	FB_SelectArray(sNetID:= , hDBID:= 1, cbCmdSize:= SIZEOF(GVL_DB.slctAllMethods), pCmdAddr:= ADR(GVL_DB.slctAllMethods), nStartIndex:= 0, nRecordCount:= 500, cbRecordArraySize:= SIZEOF(GVL_DB.listOfMethod), pDestAddr:= ADR(GVL_DB.listOfMethod), bExecute:= TRUE, tTimeout:= T#15S, bBusy=> busy, bError=> err, nErrID=> errid, sSQLState=> sqlstate, nRecords=> recAnz);
	
	IF NOT FB_SelectArray.bBusy THEN
		state:= E_DB_QUERY_STATE.IDLE_STATE;
		bExecute:= FALSE;
	ELSIF FB_SelectArray.bError THEN	
		state:= E_DB_QUERY_STATE.ERROR_STATE;
	ELSE
		state:= E_DB_QUERY_STATE.SELECT_ALL_METHODS;
		bExecute:= FALSE;
	END_IF
	
E_DB_QUERY_STATE.SELECT_ALL_ACTV_METHODS:
	
	FB_SelectArray(sNetID:= , hDBID:= 1, cbCmdSize:= SIZEOF(GVL_DB.slctAllActvMethod), pCmdAddr:= ADR(GVL_DB.slctAllActvMethod), nStartIndex:= 0, nRecordCount:= 500, cbRecordArraySize:= SIZEOF(GVL_DB.listOfMethod), pDestAddr:= ADR(GVL_DB.listOfMethod), bExecute:= TRUE, tTimeout:= T#15S, bBusy=> busy, bError=> err, nErrID=> errid, sSQLState=> sqlstate, nRecords=> recAnz);
	
	IF NOT FB_SelectArray.bBusy THEN
		state:= E_DB_QUERY_STATE.IDLE_STATE;
		bExecute:= FALSE;
	ELSIF FB_SelectArray.bError THEN	
		state:= E_DB_QUERY_STATE.ERROR_STATE;
	ELSE
		state:= E_DB_QUERY_STATE.SELECT_ALL_ACTV_METHODS;
		bExecute:= FALSE;
	END_IF
	
E_DB_QUERY_STATE.SELECT_WHOLE_METHODS:
	
	cmdSlc:= GVL_DB.slctMethod;
	selectMethod(start:=TRUE, methodName:= GVL_DB.methodName, methodRevision:= GVL_DB.methodRevision);
	FB_SelectArray(sNetID:= , hDBID:= 1, cbCmdSize:= SIZEOF(cmdSlc), pCmdAddr:= ADR(cmdSlc), nStartIndex:= 0, nRecordCount:= 26, cbRecordArraySize:= SIZEOF(GVL_DB.stParameter_MR), pDestAddr:= ADR(GVL_DB.stParameter_MR), bExecute:= TRUE, tTimeout:= T#15S, bBusy=> busy, bError=> err, nErrID=> errid, sSQLState=> sqlstate, nRecords=> recAnz);
	
	IF NOT FB_SelectArray.bBusy THEN
		timerVD(in:= TRUE, pt:= T#3S);
		bExecute:= FALSE;
		state:= E_DB_QUERY_STATE.IDLE_STATE;
	ELSIF FB_SelectArray.bError THEN	
		state:= E_DB_QUERY_STATE.ERROR_STATE;
	ELSE
		state:= E_DB_QUERY_STATE.SELECT_WHOLE_METHODS;
		bExecute:= FALSE;
	END_IF
	
E_DB_QUERY_STATE.INSERT_NEW_METHOD:

	cmdIn:= GVL_DB.isrtNewMethod;
	insertMethod(start:=TRUE);
	FB_Insert(sNetID:= , hDBID:= 1, cbCmdSize:= SIZEOF(cmdIn), pCmdAddr:= ADR(cmdIn), bExecute:= TRUE, tTimeout:= T#15S, bBusy=> busy, bError=> err, nErrID=> errid, sSQLState=> sqlstate);
	
	IF NOT FB_Insert.bBusy THEN
		state:= E_DB_QUERY_STATE.IDLE_STATE;
		bExecuteIn:= FALSE;
	ELSIF FB_Insert.bError THEN	
		state:= E_DB_QUERY_STATE.ERROR_STATE;
	ELSE
		state:= E_DB_QUERY_STATE.INSERT_NEW_METHOD;
		//bExecuteIn:= FALSE;
	END_IF	

E_DB_QUERY_STATE.UPDATE_DEACTV_METHOD:

	cmdIn:= GVL_DB.updtDactvMethod;
	updateMethod(start:=TRUE, methodName:= GVL_Recipe.stCurrentRecipe.stInfo.sMethodName, methodRevision:= INT_TO_STRING(GVL_Recipe.stCurrentRecipe.stInfo.iRevision));
	FB_Insert(sNetID:= , hDBID:= 1, cbCmdSize:= SIZEOF(cmdIn), pCmdAddr:= ADR(cmdIn), bExecute:= TRUE, tTimeout:= T#15S, bBusy=> busy, bError=> err, nErrID=> errid, sSQLState=> sqlstate);
	
	IF NOT FB_Insert.bBusy THEN
		state:= E_DB_QUERY_STATE.IDLE_STATE;
		bExecuteIn:= FALSE;
	ELSIF FB_Insert.bError THEN	
		state:= E_DB_QUERY_STATE.ERROR_STATE;
	ELSE
		state:= E_DB_QUERY_STATE.UPDATE_DEACTV_METHOD;
		//bExecuteIn:= FALSE;
	END_IF	

E_DB_QUERY_STATE.SELECT_LAST_METHOD_ID:
	
	cmdSlc:= GVL_DB.slctMethodID;
	selectMethodID(start:= TRUE, methodName:= GVL_HMI.stRecipeInfo.sMethodName);
	FB_SelectArray(sNetID:= , hDBID:= 1, cbCmdSize:= SIZEOF(cmdSlc), pCmdAddr:= ADR(cmdSlc), nStartIndex:= 0, nRecordCount:= 1, cbRecordArraySize:= SIZEOF(GVL_DB.lastMethodID), pDestAddr:= ADR(GVL_DB.lastMethodID), bExecute:= TRUE, tTimeout:= T#15S, bBusy=> busy, bError=> err, nErrID=> errid, sSQLState=> sqlstate, nRecords=> recAnz);
	
	IF NOT FB_SelectArray.bBusy THEN
		state:= E_DB_QUERY_STATE.IDLE_STATE;
		bExecute:= FALSE;
	ELSIF FB_SelectArray.bError THEN	
		state:= E_DB_QUERY_STATE.ERROR_STATE;
	ELSE
		state:= E_DB_QUERY_STATE.SELECT_LAST_METHOD_ID;
		bExecute:= FALSE;
	END_IF
	
E_DB_QUERY_STATE.SELECT_VOLUME_DATA:
	
	cmdSlc:= GVL_DB.slctVD;
	selectVD(start:=TRUE, methodID:= INT_TO_STRING(GVL_DB.stParameter_MR.methodID));
	FB_SelectArray(sNetID:= , hDBID:= 1, cbCmdSize:= SIZEOF(cmdSlc), pCmdAddr:= ADR(cmdSlc), nStartIndex:= 0, nRecordCount:= 10, cbRecordArraySize:= SIZEOF(GVL_DB.astVolData), pDestAddr:= ADR(GVL_DB.astVolData), bExecute:= TRUE, tTimeout:= T#15S, bBusy=> busy, bError=> err, nErrID=> errid, sSQLState=> sqlstate, nRecords=> recAnz);
	
	IF NOT FB_SelectArray.bBusy AND timerVD.Q THEN
		state:= E_DB_QUERY_STATE.IDLE_STATE;
		bExecute:= FALSE;
		//timerVD(in:= FALSE);
	ELSIF FB_SelectArray.bError THEN	
		state:= E_DB_QUERY_STATE.ERROR_STATE;
	ELSE
		state:= E_DB_QUERY_STATE.SELECT_VOLUME_DATA;
		bExecute:= FALSE;
	END_IF
	
E_DB_QUERY_STATE.INSERT_VOLUME_DATA:

	cmdIn:= GVL_DB.isrtVD;
	insertVD(start:=TRUE, methodID:= INT_TO_STRING(GVL_DB.lastMethodID), line:= j);
	FB_Insert(sNetID:= , hDBID:= 1, cbCmdSize:= SIZEOF(cmdIn), pCmdAddr:= ADR(cmdIn), bExecute:= TRUE, tTimeout:= T#15S, bBusy=> busy, bError=> err, nErrID=> errid, sSQLState=> sqlstate);
	
	IF NOT FB_Insert.bBusy THEN
		state:= E_DB_QUERY_STATE.IDLE_STATE;
		bExecuteIn:= FALSE;
	ELSIF FB_Insert.bError THEN	
		state:= E_DB_QUERY_STATE.ERROR_STATE;
	ELSE
		state:= E_DB_QUERY_STATE.INSERT_VOLUME_DATA;
		//bExecuteIn:= FALSE;
	END_IF	
	
E_DB_QUERY_STATE.INSERT_USER:

    cmdIn := GVL_DB.isrtUser;
    insertUser(start := TRUE, line := i);

    FB_Insert(
        sNetID := ,
        hDBID := 1,
        cbCmdSize := SIZEOF(cmdIn),
        pCmdAddr := ADR(cmdIn),
        bExecute := TRUE,
        tTimeout := T#15S,
        bBusy => busy,
        bError => err,
        nErrID => errid,
        sSQLState => sqlstate
    );

    IF NOT FB_Insert.bBusy THEN
        state := E_DB_QUERY_STATE.IDLE_STATE;
        bExecuteIn := FALSE;
    ELSIF FB_Insert.bError THEN
        state := E_DB_QUERY_STATE.ERROR_STATE;
    ELSE
        state := E_DB_QUERY_STATE.INSERT_USER;
    END_IF
(*	
E_DB_QUERY_STATE.INSERT_USER_MGMT_HISTORY:

    cmdIn := GVL_DB.isrtUserMgmtHistory;
    insertUserMgmtHistory(start := TRUE);

    GVL_HMI.stUserMgmtHistoryEvent.bBusy := TRUE;
    GVL_HMI.stUserMgmtHistoryEvent.bDone := FALSE;
    GVL_HMI.stUserMgmtHistoryEvent.bError := FALSE;
    GVL_HMI.stUserMgmtHistoryEvent.sErrorText := '';

    FB_Insert(
        sNetID := ,
        hDBID := 1,
        cbCmdSize := SIZEOF(cmdIn),
        pCmdAddr := ADR(cmdIn),
        bExecute := TRUE,
        tTimeout := T#15S,
        bBusy => busy,
        bError => err,
        nErrID => errid,
        sSQLState => sqlstate
    );

    IF NOT FB_Insert.bBusy THEN

        GVL_HMI.stUserMgmtHistoryEvent.bExecute := FALSE;
        GVL_HMI.stUserMgmtHistoryEvent.bBusy := FALSE;
        GVL_HMI.stUserMgmtHistoryEvent.bDone := TRUE;
        GVL_HMI.stUserMgmtHistoryEvent.bError := FALSE;

        state := E_DB_QUERY_STATE.IDLE_STATE;
        bExecuteIn := FALSE;

    ELSIF FB_Insert.bError THEN

        GVL_HMI.stUserMgmtHistoryEvent.bExecute := FALSE;
        GVL_HMI.stUserMgmtHistoryEvent.bBusy := FALSE;
        GVL_HMI.stUserMgmtHistoryEvent.bDone := FALSE;
        GVL_HMI.stUserMgmtHistoryEvent.bError := TRUE;
        GVL_HMI.stUserMgmtHistoryEvent.sErrorText := 'Error inserting user management history.';

        state := E_DB_QUERY_STATE.ERROR_STATE;

    ELSE

        state := E_DB_QUERY_STATE.INSERT_USER_MGMT_HISTORY;
        bExecuteIn := FALSE;

    END_IF
*)
E_DB_QUERY_STATE.SELECT_ALL_CURRENT_USERS:
	
	cmdSlc:= GVL_DB.slctCurrentUser;
	FB_SelectArray(sNetID:= , hDBID:= 1, cbCmdSize:= SIZEOF(cmdSlc), pCmdAddr:= ADR(cmdSlc), nStartIndex:= 0, nRecordCount:= 500, cbRecordArraySize:= SIZEOF(GVL_DB.astData_CUL), pDestAddr:= ADR(GVL_DB.astData_CUL), bExecute:= TRUE, tTimeout:= T#15S, bBusy=> busy, bError=> err, nErrID=> errid, sSQLState=> sqlstate, nRecords=> recAnz);
	
	IF NOT FB_SelectArray.bBusy THEN
		state:= E_DB_QUERY_STATE.IDLE_STATE;
		bExecute:= FALSE;
	ELSIF FB_SelectArray.bError THEN	
		state:= E_DB_QUERY_STATE.ERROR_STATE;
	ELSE
		state:= E_DB_QUERY_STATE.SELECT_ALL_CURRENT_USERS;
		bExecute:= FALSE;
	END_IF
	
E_DB_QUERY_STATE.SELECT_ALL_USERS:
	
	cmdSlc:= GVL_DB.slctAllUsers;
	FB_SelectArray(sNetID:= , hDBID:= 1, cbCmdSize:= SIZEOF(cmdSlc), pCmdAddr:= ADR(cmdSlc), nStartIndex:= 0, nRecordCount:= 1000, cbRecordArraySize:= SIZEOF(GVL_DB.astData_CUL), pDestAddr:= ADR(GVL_DB.astData_CUL), bExecute:= TRUE, tTimeout:= T#15S, bBusy=> busy, bError=> err, nErrID=> errid, sSQLState=> sqlstate, nRecords=> recAnz);
	
	IF NOT FB_SelectArray.bBusy THEN
		state:= E_DB_QUERY_STATE.IDLE_STATE;
		bExecute:= FALSE;
	ELSIF FB_SelectArray.bError THEN	
		state:= E_DB_QUERY_STATE.ERROR_STATE;
	ELSE
		state:= E_DB_QUERY_STATE.SELECT_ALL_USERS;
		bExecute:= FALSE;
	END_IF
	
E_DB_QUERY_STATE.SELECT_LAST_SOLVENT:
	
	cmdSlc:= GVL_DB.slctSolvent;

	FB_SelectArray(
		sNetID:= ,
		hDBID:= 1,
		cbCmdSize:= SIZEOF(cmdSlc),
		pCmdAddr:= ADR(cmdSlc),
		nStartIndex:= 0,
		nRecordCount:= 1,
		cbRecordArraySize:= SIZEOF(GVL_DB.stSolvents),
		pDestAddr:= ADR(GVL_DB.stSolvents),
		bExecute:= TRUE,
		tTimeout:= T#15S,
		bBusy=> busy,
		bError=> err,
		nErrID=> errid,
		sSQLState=> sqlstate,
		nRecords=> recAnz
	);
	
	IF NOT FB_SelectArray.bBusy THEN
		state:= E_DB_QUERY_STATE.IDLE_STATE;
		bExecute:= FALSE;

	ELSIF FB_SelectArray.bError THEN	
		state:= E_DB_QUERY_STATE.ERROR_STATE;

	ELSE
		state:= E_DB_QUERY_STATE.SELECT_LAST_SOLVENT;
		bExecute:= FALSE;
	END_IF
	
E_DB_QUERY_STATE.SELECT_ALL_SOLVENT:
	
	cmdSlc:= GVL_DB.slctAllSolvents;
	FB_SelectArray(sNetID:= , hDBID:= 1, cbCmdSize:= SIZEOF(cmdSlc), pCmdAddr:= ADR(cmdSlc), nStartIndex:= 0, nRecordCount:= 500, cbRecordArraySize:= SIZEOF(GVL_DB.listSolvents), pDestAddr:= ADR(GVL_DB.listSolvents), bExecute:= TRUE, tTimeout:= T#15S, bBusy=> busy, bError=> err, nErrID=> errid, sSQLState=> sqlstate, nRecords=> recAnz);
	
	IF NOT FB_SelectArray.bBusy THEN
		state:= E_DB_QUERY_STATE.IDLE_STATE;
		bExecute:= FALSE;
	ELSIF FB_SelectArray.bError THEN	
		state:= E_DB_QUERY_STATE.ERROR_STATE;
	ELSE
		state:= E_DB_QUERY_STATE.SELECT_ALL_SOLVENT;
		bExecute:= FALSE;
	END_IF
	
E_DB_QUERY_STATE.INSERT_SOLVENT:

	cmdIn:= GVL_DB.isrtSolvent;
	insertSolvent(start:=TRUE);
	FB_Insert(sNetID:= , hDBID:= 1, cbCmdSize:= SIZEOF(cmdIn), pCmdAddr:= ADR(cmdIn), bExecute:= TRUE, tTimeout:= T#15S, bBusy=> busy, bError=> err, nErrID=> errid, sSQLState=> sqlstate);
	
	IF NOT FB_Insert.bBusy THEN
		state:= E_DB_QUERY_STATE.IDLE_STATE;
		bExecuteIn:= FALSE;
	ELSIF FB_Insert.bError THEN	
		state:= E_DB_QUERY_STATE.ERROR_STATE;
	ELSE
		state:= E_DB_QUERY_STATE.INSERT_SOLVENT;
	END_IF	

E_DB_QUERY_STATE.INSERT_LINEAR_MOTORS:

	cmdIn:= GVL_DB.isrtLinear;
	insertLinearMotors(start:=TRUE);
	FB_Insert(sNetID:= , hDBID:= 1, cbCmdSize:= SIZEOF(cmdIn), pCmdAddr:= ADR(cmdIn), bExecute:= TRUE, tTimeout:= T#15S, bBusy=> busy, bError=> err, nErrID=> errid, sSQLState=> sqlstate);
	
	IF NOT FB_Insert.bBusy THEN
		state:= E_DB_QUERY_STATE.IDLE_STATE;
		bExecuteIn:= FALSE;
	ELSIF FB_Insert.bError THEN	
		state:= E_DB_QUERY_STATE.ERROR_STATE;
	ELSE
		state:= E_DB_QUERY_STATE.INSERT_LINEAR_MOTORS;
	END_IF
	
E_DB_QUERY_STATE.SELECT_LINEAR_MOTORS:
	
	cmdSlc:= GVL_DB.slctLinear;
	FB_SelectArray(sNetID:= , hDBID:= 1, cbCmdSize:= SIZEOF(cmdSlc), pCmdAddr:= ADR(cmdSlc), nStartIndex:= 0, nRecordCount:= 500, cbRecordArraySize:= SIZEOF(GVL_DB.stLinearMotors), pDestAddr:= ADR(GVL_DB.stLinearMotors), bExecute:= TRUE, tTimeout:= T#15S, bBusy=> busy, bError=> err, nErrID=> errid, sSQLState=> sqlstate, nRecords=> recAnz);
	
	IF NOT FB_SelectArray.bBusy THEN
		state:= E_DB_QUERY_STATE.IDLE_STATE;
		bExecute:= FALSE;
	ELSIF FB_SelectArray.bError THEN	
		state:= E_DB_QUERY_STATE.ERROR_STATE;
	ELSE
		state:= E_DB_QUERY_STATE.SELECT_LINEAR_MOTORS;
		bExecute:= FALSE;
	END_IF
	
E_DB_QUERY_STATE.SELECT_CALIB_REPORT_LIST: 
    
	GVL_Reports.bSearchBusy   := TRUE;
    GVL_Reports.bSearchDone   := FALSE;
    GVL_Reports.bSearchError  := FALSE;
    GVL_Reports.sSearchStatus := 'Loading calibration reports...';

    IF NOT bInitSelectCalibReportList THEN
        bInitSelectCalibReportList := TRUE;

        IF GVL_Reports.bUseDateFilter THEN
            selectCalibReportListByDate(
                start := TRUE,
                dateFrom := GVL_Reports.sDateFromFilter,
                dateTo := GVL_Reports.sDateToFilter
            );
        ELSE
            cmdSlc := GVL_DB.slctCalibReportListFromValues;
        END_IF

        bExecute := TRUE;
    ELSE
        bExecute := FALSE;
    END_IF

    FB_SelectArray(	sNetID:= ,
					hDBID:= 1,
					cbCmdSize:= SIZEOF(cmdSlc),
					pCmdAddr:= ADR(cmdSlc),
					nStartIndex:= 0,
					nRecordCount:= 100,
					cbRecordArraySize:= SIZEOF(GVL_Reports.aReportSearchResult),
					pDestAddr:= ADR(GVL_Reports.aReportSearchResult),
					bExecute:= TRUE,
					tTimeout:= T#15S,
					bBusy=> busy,
					bError=> err,
					nErrID=> errid,
					sSQLState=> sqlstate,
					nRecords=> recAnz);

    IF NOT FB_SelectArray.bBusy THEN
        GVL_Reports.uiReportSearchCount := recAnz;
        GVL_Reports.bSearchBusy   := FALSE;
        GVL_Reports.bSearchDone   := TRUE;
        GVL_Reports.bSearchError  := FALSE;
        GVL_Reports.sSearchStatus := 'Calibration reports loaded';
        bExecute := FALSE;
        state := E_DB_QUERY_STATE.IDLE_STATE;

    ELSIF FB_SelectArray.bError THEN
        GVL_Reports.bSearchBusy   := FALSE;
        GVL_Reports.bSearchDone   := FALSE;
        GVL_Reports.bSearchError  := TRUE;
        GVL_Reports.sSearchStatus := 'Error loading calibration reports';
        state := E_DB_QUERY_STATE.ERROR_STATE;

    ELSE
        state := E_DB_QUERY_STATE.SELECT_CALIB_REPORT_LIST;
        bExecute := FALSE;
    END_IF
	
E_DB_QUERY_STATE.SELECT_CALIB_REPORT_BY_ID:
	
	GVL_Reports.bLoadBusy   := TRUE;
    GVL_Reports.bLoadDone   := FALSE;
    GVL_Reports.bLoadError  := FALSE;
    GVL_Reports.sLoadStatus := 'Loading calibration report header...';

    IF NOT bInitSelectCalibReportByID THEN
        bInitSelectCalibReportByID := TRUE;
        Clear_PumpCalibReportBuffers();
        selectCalibReportHeaderByID(start := TRUE, calibrationID := GVL_Reports.sSelectedPrimaryID);
        bExecute := TRUE;
    ELSE
        bExecute := FALSE;
    END_IF

    FB_SelectArray(
        sNetID := ,
        hDBID := 1,
        cbCmdSize := SIZEOF(cmdSlc),
        pCmdAddr := ADR(cmdSlc),
        nStartIndex := 0,
        nRecordCount := 1,
        cbRecordArraySize := SIZEOF(GVL_Reports.aSelectedCalibReportHeader),
        pDestAddr := ADR(GVL_Reports.aSelectedCalibReportHeader),
        bExecute := bExecute,
        tTimeout := T#15S,
        bBusy => busy,
        bError => err,
        nErrID => errid,
        sSQLState => sqlstate,
        nRecords => recAnz
    );

    IF FB_SelectArray.bError THEN
        bInitSelectCalibReportByID := FALSE;
        GVL_Reports.bLoadBusy   := FALSE;
        GVL_Reports.bLoadDone   := FALSE;
        GVL_Reports.bLoadError  := TRUE;
        GVL_Reports.sLoadStatus := 'Error loading calibration report header';
        state := E_DB_QUERY_STATE.ERROR_STATE;

    ELSIF NOT FB_SelectArray.bBusy AND bInitSelectCalibReportByID THEN
        bInitSelectCalibReportByID := FALSE;

        IF recAnz > 0 THEN
			GVL_Reports.stSelectedCalibReportHeader := GVL_Reports.aSelectedCalibReportHeader[1];
            CopySelectedCalibHeaderToLegacy();
            state := E_DB_QUERY_STATE.SELECT_CALIB_REPORT_VALUES_BY_ID;
        ELSE
            GVL_Reports.bLoadBusy   := FALSE;
            GVL_Reports.bLoadDone   := FALSE;
            GVL_Reports.bLoadError  := TRUE;
            GVL_Reports.sLoadStatus := 'Calibration report header not found';
            state := E_DB_QUERY_STATE.IDLE_STATE;
        END_IF
    END_IF
	
E_DB_QUERY_STATE.SELECT_CALIB_REPORT_VALUES_BY_ID:

	GVL_Reports.bLoadBusy   := TRUE;
    GVL_Reports.bLoadDone   := FALSE;
    GVL_Reports.bLoadError  := FALSE;
    GVL_Reports.sLoadStatus := 'Loading calibration report values...';

    IF NOT bInitSelectCalibReportValuesByID THEN
        bInitSelectCalibReportValuesByID := TRUE;
        selectCalibReportValuesByID(start := TRUE, calibrationID := GVL_Reports.sSelectedPrimaryID);
        bExecute := TRUE;
    ELSE
        bExecute := FALSE;
    END_IF

    FB_SelectArray(
        sNetID := ,
        hDBID := 1,
        cbCmdSize := SIZEOF(cmdSlc),
        pCmdAddr := ADR(cmdSlc),
        nStartIndex := 0,
        nRecordCount := 300,
        cbRecordArraySize := SIZEOF(GVL_Reports.aSelectedCalibReportLines),
        pDestAddr := ADR(GVL_Reports.aSelectedCalibReportLines),
        bExecute := bExecute,
        tTimeout := T#15S,
        bBusy => busy,
        bError => err,
        nErrID => errid,
        sSQLState => sqlstate,
        nRecords => recAnz
    );

    IF FB_SelectArray.bError THEN
        bInitSelectCalibReportValuesByID := FALSE;
        GVL_Reports.bLoadBusy   := FALSE;
        GVL_Reports.bLoadDone   := FALSE;
        GVL_Reports.bLoadError  := TRUE;
        GVL_Reports.sLoadStatus := 'Error loading calibration report values';
        state := E_DB_QUERY_STATE.ERROR_STATE;

    ELSIF NOT FB_SelectArray.bBusy AND bInitSelectCalibReportValuesByID THEN
        bInitSelectCalibReportValuesByID := FALSE;
		
		CopySelectedCalibLinesToLegacy();

        GVL_Reports.bLoadBusy      := FALSE;
        GVL_Reports.bLoadDone      := TRUE;
        GVL_Reports.bLoadError     := FALSE;
        GVL_Reports.bPdfDataReady  := TRUE;
        GVL_Reports.bPdfConsumed   := FALSE;
        GVL_Reports.sLoadStatus    := 'Calibration report loaded';

        state := E_DB_QUERY_STATE.IDLE_STATE;
    END_IF
	
E_DB_QUERY_STATE.SELECT_SYSTEM_SETTINGS_REPORT_LIST:

	GVL_Reports.bSearchBusy   := TRUE;
    GVL_Reports.bSearchDone   := FALSE;
    GVL_Reports.bSearchError  := FALSE;
    GVL_Reports.sSearchStatus := 'Loading system settings reports...';

    IF NOT bInitSelectSystemSettingsReportList THEN
        bInitSelectSystemSettingsReportList := TRUE;

        IF GVL_Reports.bUseDateFilter THEN
            selectSystemSettingsReportListByDate(
                start := TRUE,
                dateFrom := GVL_Reports.sDateFromFilter,
                dateTo := GVL_Reports.sDateToFilter
            );
        ELSE
            cmdSlc := GVL_DB.slctSystemSettingsReportList;
        END_IF

        bExecute := TRUE;
    ELSE
        bExecute := FALSE;
    END_IF

    FB_SelectArray(
        sNetID := ,
        hDBID := 1,
        cbCmdSize := SIZEOF(cmdSlc),
        pCmdAddr := ADR(cmdSlc),
        nStartIndex := 0,
        nRecordCount := 100,
        cbRecordArraySize := SIZEOF(GVL_Reports.aReportSearchResult),
        pDestAddr := ADR(GVL_Reports.aReportSearchResult),
        bExecute := bExecute,
        tTimeout := T#15S,
        bBusy => busy,
        bError => err,
        nErrID => errid,
        sSQLState => sqlstate,
        nRecords => recAnz
    );

    IF FB_SelectArray.bError THEN
        bInitSelectSystemSettingsReportList := FALSE;
        GVL_Reports.bSearchBusy   := FALSE;
        GVL_Reports.bSearchDone   := FALSE;
        GVL_Reports.bSearchError  := TRUE;
        GVL_Reports.sSearchStatus := 'Error loading system settings reports';
        state := E_DB_QUERY_STATE.ERROR_STATE;

    ELSIF NOT FB_SelectArray.bBusy AND bInitSelectSystemSettingsReportList THEN
        bInitSelectSystemSettingsReportList := FALSE;
        GVL_Reports.uiReportSearchCount := recAnz;
        GVL_Reports.bSearchBusy   := FALSE;
        GVL_Reports.bSearchDone   := TRUE;
        GVL_Reports.bSearchError  := FALSE;
        GVL_Reports.sSearchStatus := 'System settings reports loaded';
        state := E_DB_QUERY_STATE.IDLE_STATE;
    END_IF
	
E_DB_QUERY_STATE.SELECT_SYSTEM_SETTINGS_BY_ID:

    GVL_Reports.bLoadBusy   := TRUE;
    GVL_Reports.bLoadDone   := FALSE;
    GVL_Reports.bLoadError  := FALSE;
    GVL_Reports.sLoadStatus := 'Loading system settings report...';

    IF NOT bInitSelectSystemSettingsByID THEN
        bInitSelectSystemSettingsByID := TRUE;
        Clear_SystemSettingsReportBuffer();
        selectSystemSettingsByID(start := TRUE, revisionID := GVL_Reports.sSelectedPrimaryID);
        bExecute := TRUE;
    ELSE
        bExecute := FALSE;
    END_IF

    FB_SelectArray(
        sNetID := ,
        hDBID := 1,
        cbCmdSize := SIZEOF(cmdSlc),
        pCmdAddr := ADR(cmdSlc),
        nStartIndex := 0,
        nRecordCount := 1,
        cbRecordArraySize := SIZEOF(GVL_Reports.aSelectedSystemSettingsBuf),
        pDestAddr := ADR(GVL_Reports.aSelectedSystemSettingsBuf),
        bExecute := bExecute,
        tTimeout := T#15S,
        bBusy => busy,
        bError => err,
        nErrID => errid,
        sSQLState => sqlstate,
        nRecords => recAnz
    );

    IF FB_SelectArray.bError THEN
        bInitSelectSystemSettingsByID := FALSE;
        GVL_Reports.bLoadBusy   := FALSE;
        GVL_Reports.bLoadDone   := FALSE;
        GVL_Reports.bLoadError  := TRUE;
        GVL_Reports.sLoadStatus := 'Error loading system settings report';
        state := E_DB_QUERY_STATE.ERROR_STATE;

    ELSIF NOT FB_SelectArray.bBusy AND bInitSelectSystemSettingsByID THEN
        bInitSelectSystemSettingsByID := FALSE;

        IF recAnz > 0 THEN
            GVL_Reports.stSelectedSystemSettings := GVL_Reports.aSelectedSystemSettingsBuf[1];
            GVL_Reports.bLoadBusy      := FALSE;
            GVL_Reports.bLoadDone      := TRUE;
            GVL_Reports.bLoadError     := FALSE;
            GVL_Reports.bPdfDataReady  := TRUE;
            GVL_Reports.bPdfConsumed   := FALSE;
            GVL_Reports.sLoadStatus    := 'System settings report loaded';
            state := E_DB_QUERY_STATE.IDLE_STATE;
        ELSE
            GVL_Reports.bLoadBusy   := FALSE;
            GVL_Reports.bLoadDone   := FALSE;
            GVL_Reports.bLoadError  := TRUE;
            GVL_Reports.sLoadStatus := 'System settings report not found';
            state := E_DB_QUERY_STATE.IDLE_STATE;
        END_IF
    END_IF

E_DB_QUERY_STATE.SELECT_METHOD_REPORT_LIST:

    GVL_Reports.bSearchBusy   := TRUE;
    GVL_Reports.bSearchDone   := FALSE;
    GVL_Reports.bSearchError  := FALSE;
    GVL_Reports.sSearchStatus := 'Loading method list...';

    IF NOT bInitSelectMethodReportList THEN
        bInitSelectMethodReportList := TRUE;
        cmdSlc := GVL_DB.slctMethodReportList;
        bExecute := TRUE;
    ELSE
        bExecute := FALSE;
    END_IF

    FB_SelectArray(
        sNetID            := ,
        hDBID             := 1,
        cbCmdSize         := SIZEOF(cmdSlc),
        pCmdAddr          := ADR(cmdSlc),
        nStartIndex       := 0,
        nRecordCount      := 100,
        cbRecordArraySize := SIZEOF(GVL_Reports.aReportSearchResult),
        pDestAddr         := ADR(GVL_Reports.aReportSearchResult),
        bExecute          := bExecute,
        tTimeout          := T#15S,
        bBusy             => busy,
        bError            => err,
        nErrID            => errid,
        sSQLState         => sqlstate,
        nRecords          => recAnz
    );

    IF NOT FB_SelectArray.bBusy THEN
        bInitSelectMethodReportList       := FALSE;
        GVL_Reports.uiReportSearchCount   := recAnz;
        GVL_Reports.bSearchBusy           := FALSE;
        GVL_Reports.bSearchDone           := TRUE;
        GVL_Reports.bSearchError          := FALSE;
        GVL_Reports.sSearchStatus         := 'Method list loaded';
        bExecute := FALSE;
        state := E_DB_QUERY_STATE.IDLE_STATE;

    ELSIF FB_SelectArray.bError THEN
        bInitSelectMethodReportList  := FALSE;
        GVL_Reports.bSearchBusy      := FALSE;
        GVL_Reports.bSearchDone      := FALSE;
        GVL_Reports.bSearchError     := TRUE;
        GVL_Reports.sSearchStatus    := 'Error loading method list';
        state := E_DB_QUERY_STATE.ERROR_STATE;

    ELSE
        state    := E_DB_QUERY_STATE.SELECT_METHOD_REPORT_LIST;
        bExecute := FALSE;
    END_IF
	
// Report search - latest revision per method, supports date filter
E_DB_QUERY_STATE.SELECT_METHOD_REPORT_SEARCH:

    GVL_Reports.bSearchBusy   := TRUE;
    GVL_Reports.bSearchDone   := FALSE;
    GVL_Reports.bSearchError  := FALSE;
    GVL_Reports.sSearchStatus := 'Loading method reports...';

    IF NOT bInitSelectMethodReportSearch THEN
        bInitSelectMethodReportSearch := TRUE;

        IF GVL_Reports.bUseDateFilter THEN
            selectMethodReportSearchByDate(
                start    := TRUE,
                dateFrom := GVL_Reports.sDateFromFilter,
                dateTo   := GVL_Reports.sDateToFilter
            );
        ELSE
            cmdSlc := GVL_DB.slctMethodReportSearchLatest;
        END_IF

        bExecute := TRUE;
    ELSE
        bExecute := FALSE;
    END_IF

    FB_SelectArray(
        sNetID            := ,
        hDBID             := 1,
        cbCmdSize         := SIZEOF(cmdSlc),
        pCmdAddr          := ADR(cmdSlc),
        nStartIndex       := 0,
        nRecordCount      := 100,
        cbRecordArraySize := SIZEOF(GVL_Reports.aReportSearchResult),
        pDestAddr         := ADR(GVL_Reports.aReportSearchResult),
        bExecute          := bExecute,
        tTimeout          := T#15S,
        bBusy             => busy,
        bError            => err,
        nErrID            => errid,
        sSQLState         => sqlstate,
        nRecords          => recAnz
    );

    IF FB_SelectArray.bError THEN
        bInitSelectMethodReportSearch := FALSE;
        GVL_Reports.bSearchBusy       := FALSE;
        GVL_Reports.bSearchDone       := FALSE;
        GVL_Reports.bSearchError      := TRUE;
        GVL_Reports.sSearchStatus     := 'Error loading method reports';
        state := E_DB_QUERY_STATE.ERROR_STATE;

    ELSIF NOT FB_SelectArray.bBusy AND bInitSelectMethodReportSearch THEN
        bInitSelectMethodReportSearch := FALSE;
        GVL_Reports.uiReportSearchCount := recAnz;
        GVL_Reports.bSearchBusy       := FALSE;
        GVL_Reports.bSearchDone       := TRUE;
        GVL_Reports.bSearchError      := FALSE;
        GVL_Reports.sSearchStatus     := 'Method reports loaded';
        state := E_DB_QUERY_STATE.IDLE_STATE;

    ELSE
        state := E_DB_QUERY_STATE.SELECT_METHOD_REPORT_SEARCH;
    END_IF

E_DB_QUERY_STATE.SELECT_RUN_REPORT_LIST:

    GVL_Reports.bSearchBusy   := TRUE;
    GVL_Reports.bSearchDone   := FALSE;
    GVL_Reports.bSearchError  := FALSE;
    GVL_Reports.sSearchStatus := 'Loading run reports...';

    IF NOT bInitSelectRunReportList THEN
        bInitSelectRunReportList := TRUE;
        cmdSlc := GVL_DB.slctRunReportList;
        bExecute := TRUE;
    ELSE
        bExecute := FALSE;
    END_IF

    FB_SelectArray(
        sNetID            := ,
        hDBID             := 1,
        cbCmdSize         := SIZEOF(cmdSlc),
        pCmdAddr          := ADR(cmdSlc),
        nStartIndex       := 0,
        nRecordCount      := 100,
        cbRecordArraySize := SIZEOF(GVL_Reports.aReportSearchResult),
        pDestAddr         := ADR(GVL_Reports.aReportSearchResult),
        bExecute          := bExecute,
        tTimeout          := T#15S,
        bBusy             => busy,
        bError            => err,
        nErrID            => errid,
        sSQLState         => sqlstate,
        nRecords          => recAnz
    );

    IF NOT FB_SelectArray.bBusy THEN
        bInitSelectRunReportList          := FALSE;
        GVL_Reports.uiReportSearchCount   := recAnz;
        GVL_Reports.bSearchBusy           := FALSE;
        GVL_Reports.bSearchDone           := TRUE;
        GVL_Reports.bSearchError          := FALSE;
        GVL_Reports.sSearchStatus         := 'Run reports loaded';
        bExecute := FALSE;
        state := E_DB_QUERY_STATE.IDLE_STATE;

    ELSIF FB_SelectArray.bError THEN
        bInitSelectRunReportList := FALSE;
        GVL_Reports.bSearchBusy  := FALSE;
        GVL_Reports.bSearchDone  := FALSE;
        GVL_Reports.bSearchError := TRUE;
        GVL_Reports.sSearchStatus := 'Error loading run reports';
        state := E_DB_QUERY_STATE.ERROR_STATE;

    ELSE
        state    := E_DB_QUERY_STATE.SELECT_RUN_REPORT_LIST;
        bExecute := FALSE;
    END_IF

E_DB_QUERY_STATE.SELECT_RECIPE_HEADER_BY_ID:

    GVL_Reports.bLoadBusy   := TRUE;
    GVL_Reports.bLoadDone   := FALSE;
    GVL_Reports.bLoadError  := FALSE;
    GVL_Reports.sLoadStatus := 'Loading recipe header...';

    IF NOT bInitSelectRecipeHeaderByID THEN
        bInitSelectRecipeHeaderByID := TRUE;

        Clear_MethodReportBuffers();
        selectRecipeHeaderByID(
            start := TRUE,
            methodID := GVL_Reports.sSelectedPrimaryID
        );

        bExecute := TRUE;
    ELSE
        bExecute := FALSE;
    END_IF

    FB_SelectArray(
        sNetID := ,
        hDBID := 1,
        cbCmdSize := SIZEOF(cmdSlc),
        pCmdAddr := ADR(cmdSlc),
        nStartIndex := 0,
        nRecordCount := 1,
        cbRecordArraySize := SIZEOF(GVL_Reports.stMethodHeader),
        pDestAddr := ADR(GVL_Reports.stMethodHeader),
        bExecute := bExecute,
        tTimeout := T#15S,
        bBusy => busy,
        bError => err,
        nErrID => errid,
        sSQLState => sqlstate,
        nRecords => recAnz
    );

    IF FB_SelectArray.bError THEN
        bInitSelectRecipeHeaderByID := FALSE;
        GVL_Reports.bLoadBusy   := FALSE;
        GVL_Reports.bLoadDone   := FALSE;
        GVL_Reports.bLoadError  := TRUE;
        GVL_Reports.sLoadStatus := 'Error loading recipe header';
        state := E_DB_QUERY_STATE.ERROR_STATE;

    ELSIF NOT FB_SelectArray.bBusy AND bInitSelectRecipeHeaderByID THEN
        bInitSelectRecipeHeaderByID := FALSE;

        IF recAnz > 0 THEN
            state := E_DB_QUERY_STATE.SELECT_RECIPE_VOLUME_BY_ID;
        ELSE
            GVL_Reports.bLoadBusy   := FALSE;
            GVL_Reports.bLoadDone   := FALSE;
            GVL_Reports.bLoadError  := TRUE;
            GVL_Reports.sLoadStatus := 'Recipe not found';
            state := E_DB_QUERY_STATE.IDLE_STATE;
        END_IF

    ELSE
        state := E_DB_QUERY_STATE.SELECT_RECIPE_HEADER_BY_ID;
    END_IF	
	
E_DB_QUERY_STATE.SELECT_RECIPE_VOLUME_BY_ID:

    GVL_Reports.bLoadBusy   := TRUE;
    GVL_Reports.bLoadDone   := FALSE;
    GVL_Reports.bLoadError  := FALSE;
    GVL_Reports.sLoadStatus := 'Loading recipe volume data...';

    IF NOT bInitSelectRecipeVolumeByID THEN
        bInitSelectRecipeVolumeByID := TRUE;

        selectRecipeVolumeByID(
            start := TRUE,
            methodID := GVL_Reports.sSelectedPrimaryID
        );

        bExecute := TRUE;
    ELSE
        bExecute := FALSE;
    END_IF

    FB_SelectArray(
        sNetID := ,
        hDBID := 1,
        cbCmdSize := SIZEOF(cmdSlc),
        pCmdAddr := ADR(cmdSlc),
        nStartIndex := 0,
        nRecordCount := 10,
        cbRecordArraySize := SIZEOF(GVL_Reports.aMethodVolumeData),
        pDestAddr := ADR(GVL_Reports.aMethodVolumeData),
        bExecute := bExecute,
        tTimeout := T#15S,
        bBusy => busy,
        bError => err,
        nErrID => errid,
        sSQLState => sqlstate,
        nRecords => recAnz
    );

    IF FB_SelectArray.bError THEN
        bInitSelectRecipeVolumeByID := FALSE;
        GVL_Reports.bLoadBusy   := FALSE;
        GVL_Reports.bLoadDone   := FALSE;
        GVL_Reports.bLoadError  := TRUE;
        GVL_Reports.sLoadStatus := 'Error loading recipe volume data';
        state := E_DB_QUERY_STATE.ERROR_STATE;

    ELSIF NOT FB_SelectArray.bBusy AND bInitSelectRecipeVolumeByID THEN
        bInitSelectRecipeVolumeByID := FALSE;
        GVL_Reports.bLoadBusy      := FALSE;
        GVL_Reports.bLoadDone      := TRUE;
        GVL_Reports.bLoadError     := FALSE;
        GVL_Reports.bPdfDataReady  := TRUE;
        GVL_Reports.bPdfConsumed   := FALSE;
        GVL_Reports.sLoadStatus    := 'Recipe report loaded';
        state := E_DB_QUERY_STATE.IDLE_STATE;

    ELSE
        state := E_DB_QUERY_STATE.SELECT_RECIPE_VOLUME_BY_ID;
    END_IF
	
E_DB_QUERY_STATE.SELECT_POSTRUN_RUN_BY_ID:

    GVL_Reports.bLoadBusy   := TRUE;
    GVL_Reports.bLoadDone   := FALSE;
    GVL_Reports.bLoadError  := FALSE;
    GVL_Reports.sLoadStatus := 'Loading post run header...';

    IF NOT bInitSelectPostRunByID THEN
        bInitSelectPostRunByID := TRUE;

        Clear_PostRunBuffers();

        selectPostRunHeaderByID(
            start := TRUE,
            runID := GVL_Reports.sSelectedPrimaryID
        );

        bExecute := TRUE;
    ELSE
        bExecute := FALSE;
    END_IF

    FB_SelectArray(
        sNetID := ,
        hDBID := 1,
        cbCmdSize := SIZEOF(cmdSlc),
        pCmdAddr := ADR(cmdSlc),
        nStartIndex := 0,
        nRecordCount := 1,
        cbRecordArraySize := SIZEOF(GVL_Reports.stRunHeader),
        pDestAddr := ADR(GVL_Reports.stRunHeader),
        bExecute := bExecute,
        tTimeout := T#15S,
        bBusy => busy,
        bError => err,
        nErrID => errid,
        sSQLState => sqlstate,
        nRecords => recAnz
    );

    IF FB_SelectArray.bError THEN
        bInitSelectPostRunByID := FALSE;
        GVL_Reports.bLoadBusy   := FALSE;
        GVL_Reports.bLoadDone   := FALSE;
        GVL_Reports.bLoadError  := TRUE;
        GVL_Reports.sLoadStatus := 'Error loading post run header';
        state := E_DB_QUERY_STATE.ERROR_STATE;

    ELSIF NOT FB_SelectArray.bBusy AND bInitSelectPostRunByID THEN
        bInitSelectPostRunByID := FALSE;

        IF recAnz > 0 THEN
            sPostRunMethodID := INT_TO_STRING(GVL_Reports.stRunHeader.methodID);
            state := E_DB_QUERY_STATE.SELECT_POSTRUN_METHOD_BY_RUN_ID;
        ELSE
            GVL_Reports.bLoadBusy   := FALSE;
            GVL_Reports.bLoadDone   := FALSE;
            GVL_Reports.bLoadError  := TRUE;
            GVL_Reports.sLoadStatus := 'Post run report not found';
            state := E_DB_QUERY_STATE.IDLE_STATE;
        END_IF

    ELSE
        state := E_DB_QUERY_STATE.SELECT_POSTRUN_RUN_BY_ID;
    END_IF
	
E_DB_QUERY_STATE.SELECT_POSTRUN_METHOD_BY_RUN_ID:

    GVL_Reports.bLoadBusy   := TRUE;
    GVL_Reports.bLoadDone   := FALSE;
    GVL_Reports.bLoadError  := FALSE;
    GVL_Reports.sLoadStatus := 'Loading post run method...';

    IF NOT bInitSelectPostRunMethodByID THEN
        bInitSelectPostRunMethodByID := TRUE;

        selectPostRunMethodHeaderByID(
            start := TRUE,
            methodID := sPostRunMethodID
        );

        bExecute := TRUE;
    ELSE
        bExecute := FALSE;
    END_IF

    FB_SelectArray(
        sNetID := ,
        hDBID := 1,
        cbCmdSize := SIZEOF(cmdSlc),
        pCmdAddr := ADR(cmdSlc),
        nStartIndex := 0,
        nRecordCount := 1,
        cbRecordArraySize := SIZEOF(GVL_Reports.stRunMethodHeader),
        pDestAddr := ADR(GVL_Reports.stRunMethodHeader),
        bExecute := bExecute,
        tTimeout := T#15S,
        bBusy => busy,
        bError => err,
        nErrID => errid,
        sSQLState => sqlstate,
        nRecords => recAnz
    );

    IF FB_SelectArray.bError THEN
        bInitSelectPostRunMethodByID := FALSE;
        GVL_Reports.bLoadBusy   := FALSE;
        GVL_Reports.bLoadDone   := FALSE;
        GVL_Reports.bLoadError  := TRUE;
        GVL_Reports.sLoadStatus := 'Error loading post run method';
        state := E_DB_QUERY_STATE.ERROR_STATE;

    ELSIF NOT FB_SelectArray.bBusy AND bInitSelectPostRunMethodByID THEN
        bInitSelectPostRunMethodByID := FALSE;
        state := E_DB_QUERY_STATE.SELECT_POSTRUN_VOLUME_BY_METHOD_ID;

    ELSE
        state := E_DB_QUERY_STATE.SELECT_POSTRUN_METHOD_BY_RUN_ID;
    END_IF
	
E_DB_QUERY_STATE.SELECT_POSTRUN_VOLUME_BY_METHOD_ID:

    GVL_Reports.bLoadBusy   := TRUE;
    GVL_Reports.bLoadDone   := FALSE;
    GVL_Reports.bLoadError  := FALSE;
    GVL_Reports.sLoadStatus := 'Loading post run volume data...';

    IF NOT bInitSelectPostRunVolumeByMethodID THEN
        bInitSelectPostRunVolumeByMethodID := TRUE;

        selectPostRunVolumeByMethodID(
            start := TRUE,
            methodID := sPostRunMethodID
        );

        bExecute := TRUE;
    ELSE
        bExecute := FALSE;
    END_IF

    FB_SelectArray(
        sNetID := ,
        hDBID := 1,
        cbCmdSize := SIZEOF(cmdSlc),
        pCmdAddr := ADR(cmdSlc),
        nStartIndex := 0,
        nRecordCount := 10,
        cbRecordArraySize := SIZEOF(GVL_Reports.aRunVolumeData),
        pDestAddr := ADR(GVL_Reports.aRunVolumeData),
        bExecute := bExecute,
        tTimeout := T#15S,
        bBusy => busy,
        bError => err,
        nErrID => errid,
        sSQLState => sqlstate,
        nRecords => recAnz
    );

    IF FB_SelectArray.bError THEN
        bInitSelectPostRunVolumeByMethodID := FALSE;
        GVL_Reports.bLoadBusy   := FALSE;
        GVL_Reports.bLoadDone   := FALSE;
        GVL_Reports.bLoadError  := TRUE;
        GVL_Reports.sLoadStatus := 'Error loading post run volume data';
        state := E_DB_QUERY_STATE.ERROR_STATE;

    ELSIF NOT FB_SelectArray.bBusy AND bInitSelectPostRunVolumeByMethodID THEN
        bInitSelectPostRunVolumeByMethodID := FALSE;
        GVL_Reports.bLoadBusy      := FALSE;
        GVL_Reports.bLoadDone      := TRUE;
        GVL_Reports.bLoadError     := FALSE;
        GVL_Reports.bPdfDataReady  := TRUE;
        GVL_Reports.bPdfConsumed   := FALSE;
        GVL_Reports.sLoadStatus    := 'Post run report loaded';
        state := E_DB_QUERY_STATE.IDLE_STATE;

    ELSE
        state := E_DB_QUERY_STATE.SELECT_POSTRUN_VOLUME_BY_METHOD_ID;
    END_IF

E_DB_QUERY_STATE.SELECT_LINEAR_BY_ID:

    GVL_Reports.bLoadBusy   := TRUE;
    GVL_Reports.bLoadDone   := FALSE;
    GVL_Reports.bLoadError  := FALSE;
    GVL_Reports.sLoadStatus := 'Loading linear pumps report...';

    IF NOT bInitSelectLinearByID THEN
        bInitSelectLinearByID := TRUE;

        Clear_LinearReportBuffer();

        selectLinearByID(
            start := TRUE,
            linearID := GVL_Reports.sSelectedPrimaryID
        );

        bExecute := TRUE;
    ELSE
        bExecute := FALSE;
    END_IF

    FB_SelectArray(
        sNetID := ,
        hDBID := 1,
        cbCmdSize := SIZEOF(cmdSlc),
        pCmdAddr := ADR(cmdSlc),
        nStartIndex := 0,
        nRecordCount := 1,
        cbRecordArraySize := SIZEOF(GVL_Reports.stLinearReport),
        pDestAddr := ADR(GVL_Reports.stLinearReport),
        bExecute := bExecute,
        tTimeout := T#15S,
        bBusy => busy,
        bError => err,
        nErrID => errid,
        sSQLState => sqlstate,
        nRecords => recAnz
    );

    IF FB_SelectArray.bError THEN
        bInitSelectLinearByID := FALSE;
        GVL_Reports.bLoadBusy   := FALSE;
        GVL_Reports.bLoadDone   := FALSE;
        GVL_Reports.bLoadError  := TRUE;
        GVL_Reports.sLoadStatus := 'Error loading linear pumps report';
        state := E_DB_QUERY_STATE.ERROR_STATE;

    ELSIF NOT FB_SelectArray.bBusy AND bInitSelectLinearByID THEN
        bInitSelectLinearByID := FALSE;

        IF recAnz > 0 THEN
            GVL_Reports.bLoadBusy      := FALSE;
            GVL_Reports.bLoadDone      := TRUE;
            GVL_Reports.bLoadError     := FALSE;
            GVL_Reports.bPdfDataReady  := TRUE;
            GVL_Reports.bPdfConsumed   := FALSE;
            GVL_Reports.sLoadStatus    := 'Linear pumps report loaded';
            state := E_DB_QUERY_STATE.IDLE_STATE;
        ELSE
            GVL_Reports.bLoadBusy   := FALSE;
            GVL_Reports.bLoadDone   := FALSE;
            GVL_Reports.bLoadError  := TRUE;
            GVL_Reports.sLoadStatus := 'Linear pumps report not found';
            state := E_DB_QUERY_STATE.IDLE_STATE;
        END_IF

    ELSE
        state := E_DB_QUERY_STATE.SELECT_LINEAR_BY_ID;
    END_IF
	
E_DB_QUERY_STATE.SELECT_LINEAR_REPORT_SEARCH:

    GVL_Reports.bSearchBusy   := TRUE;
    GVL_Reports.bSearchDone   := FALSE;
    GVL_Reports.bSearchError  := FALSE;
    GVL_Reports.sSearchStatus := 'Loading linear pumps reports...';

    IF NOT bInitSelectLinearReportSearch THEN
        bInitSelectLinearReportSearch := TRUE;

        IF GVL_Reports.bUseDateFilter THEN
            selectLinearReportSearchByDate(
                start := TRUE,
                dateFrom := GVL_Reports.sDateFromFilter,
                dateTo := GVL_Reports.sDateToFilter
            );
        ELSE
            cmdSlc := GVL_DB.slctLinearReportSearch;
        END_IF

        bExecute := TRUE;
    ELSE
        bExecute := FALSE;
    END_IF

    FB_SelectArray(
        sNetID := ,
        hDBID := 1,
        cbCmdSize := SIZEOF(cmdSlc),
        pCmdAddr := ADR(cmdSlc),
        nStartIndex := 0,
        nRecordCount := 100,
        cbRecordArraySize := SIZEOF(GVL_Reports.aReportSearchResult),
        pDestAddr := ADR(GVL_Reports.aReportSearchResult),
        bExecute := bExecute,
        tTimeout := T#15S,
        bBusy => busy,
        bError => err,
        nErrID => errid,
        sSQLState => sqlstate,
        nRecords => recAnz
    );

    IF FB_SelectArray.bError THEN
        bInitSelectLinearReportSearch := FALSE;
        GVL_Reports.bSearchBusy   := FALSE;
        GVL_Reports.bSearchDone   := FALSE;
        GVL_Reports.bSearchError  := TRUE;
        GVL_Reports.sSearchStatus := 'Error loading linear pumps reports';
        state := E_DB_QUERY_STATE.ERROR_STATE;

    ELSIF NOT FB_SelectArray.bBusy AND bInitSelectLinearReportSearch THEN
        bInitSelectLinearReportSearch := FALSE;
        GVL_Reports.uiReportSearchCount := recAnz;
        GVL_Reports.bSearchBusy   := FALSE;
        GVL_Reports.bSearchDone   := TRUE;
        GVL_Reports.bSearchError  := FALSE;
        GVL_Reports.sSearchStatus := 'Linear pumps reports loaded';
        state := E_DB_QUERY_STATE.IDLE_STATE;

    ELSE
        state := E_DB_QUERY_STATE.SELECT_LINEAR_REPORT_SEARCH;
    END_IF

E_DB_QUERY_STATE.SELECT_LAST_LINEAR_REPORT:

    GVL_Reports.bLoadBusy   := TRUE;
    GVL_Reports.bLoadDone   := FALSE;
    GVL_Reports.bLoadError  := FALSE;
    GVL_Reports.sLoadStatus := 'Loading current linear pumps report...';

    IF NOT bInitSelectLastLinearReport THEN
        bInitSelectLastLinearReport := TRUE;

        Clear_LinearReportBuffer();
        cmdSlc := GVL_DB.slctLastLinear;
        bExecute := TRUE;
    ELSE
        bExecute := FALSE;
    END_IF

    FB_SelectArray(
        sNetID := ,
        hDBID := 1,
        cbCmdSize := SIZEOF(cmdSlc),
        pCmdAddr := ADR(cmdSlc),
        nStartIndex := 0,
        nRecordCount := 1,
        cbRecordArraySize := SIZEOF(GVL_Reports.stLinearReport),
        pDestAddr := ADR(GVL_Reports.stLinearReport),
        bExecute := bExecute,
        tTimeout := T#15S,
        bBusy => busy,
        bError => err,
        nErrID => errid,
        sSQLState => sqlstate,
        nRecords => recAnz
    );

    IF FB_SelectArray.bError THEN
        bInitSelectLastLinearReport := FALSE;
        GVL_Reports.bLoadBusy   := FALSE;
        GVL_Reports.bLoadDone   := FALSE;
        GVL_Reports.bLoadError  := TRUE;
        GVL_Reports.sLoadStatus := 'Error loading current linear pumps report';
        state := E_DB_QUERY_STATE.ERROR_STATE;

    ELSIF NOT FB_SelectArray.bBusy AND bInitSelectLastLinearReport THEN
        bInitSelectLastLinearReport := FALSE;

        IF recAnz > 0 THEN
            GVL_Reports.bLoadBusy      := FALSE;
            GVL_Reports.bLoadDone      := TRUE;
            GVL_Reports.bLoadError     := FALSE;
            GVL_Reports.bPdfDataReady  := TRUE;
            GVL_Reports.bPdfConsumed   := FALSE;
            GVL_Reports.sLoadStatus    := 'Current linear pumps report loaded';
            state := E_DB_QUERY_STATE.IDLE_STATE;
        ELSE
            GVL_Reports.bLoadBusy   := FALSE;
            GVL_Reports.bLoadDone   := FALSE;
            GVL_Reports.bLoadError  := TRUE;
            GVL_Reports.sLoadStatus := 'No linear pumps report found';
            state := E_DB_QUERY_STATE.IDLE_STATE;
        END_IF

    ELSE
        state := E_DB_QUERY_STATE.SELECT_LAST_LINEAR_REPORT;
    END_IF	
	
E_DB_QUERY_STATE.SELECT_LAST_POSTRUN_RUN:

    GVL_Reports.bLoadBusy   := TRUE;
    GVL_Reports.bLoadDone   := FALSE;
    GVL_Reports.bLoadError  := FALSE;
    GVL_Reports.sLoadStatus := 'Loading last post-run report...';

    IF NOT bInitSelectLastPostRunRun THEN
        bInitSelectLastPostRunRun := TRUE;

        Clear_PostRunBuffers();
        cmdSlc := GVL_DB.slctLastRun;
        bExecute := TRUE;
    ELSE
        bExecute := FALSE;
    END_IF

    FB_SelectArray(
        sNetID := ,
        hDBID := 1,
        cbCmdSize := SIZEOF(cmdSlc),
        pCmdAddr := ADR(cmdSlc),
        nStartIndex := 0,
        nRecordCount := 1,
        cbRecordArraySize := SIZEOF(GVL_Reports.stRunHeader),
        pDestAddr := ADR(GVL_Reports.stRunHeader),
        bExecute := bExecute,
        tTimeout := T#15S,
        bBusy => busy,
        bError => err,
        nErrID => errid,
        sSQLState => sqlstate,
        nRecords => recAnz
    );

    IF FB_SelectArray.bError THEN
        bInitSelectLastPostRunRun := FALSE;
        GVL_Reports.bLoadBusy   := FALSE;
        GVL_Reports.bLoadDone   := FALSE;
        GVL_Reports.bLoadError  := TRUE;
        GVL_Reports.sLoadStatus := 'Error loading last post-run report';
        state := E_DB_QUERY_STATE.ERROR_STATE;

    ELSIF NOT FB_SelectArray.bBusy AND bInitSelectLastPostRunRun THEN
        bInitSelectLastPostRunRun := FALSE;

        IF recAnz > 0 THEN
            sPostRunMethodID := INT_TO_STRING(GVL_Reports.stRunHeader.methodID);
            state := E_DB_QUERY_STATE.SELECT_POSTRUN_METHOD_BY_RUN_ID;
        ELSE
            GVL_Reports.bLoadBusy   := FALSE;
            GVL_Reports.bLoadDone   := FALSE;
            GVL_Reports.bLoadError  := TRUE;
            GVL_Reports.sLoadStatus := 'No post-run report found';
            state := E_DB_QUERY_STATE.IDLE_STATE;
        END_IF

    ELSE
        state := E_DB_QUERY_STATE.SELECT_LAST_POSTRUN_RUN;
    END_IF

E_DB_QUERY_STATE.SELECT_LAST_PUMP_CALIBRATION:

    GVL_Reports.bLoadBusy   := TRUE;
    GVL_Reports.bLoadDone   := FALSE;
    GVL_Reports.bLoadError  := FALSE;
    GVL_Reports.sLoadStatus := 'Loading last pump calibration report...';

    IF NOT bInitSelectLastPumpCalibration THEN
        bInitSelectLastPumpCalibration := TRUE;

        cmdSlc := GVL_DB.slctLastCalibID;
        bExecute := TRUE;
    ELSE
        bExecute := FALSE;
    END_IF

    FB_SelectArray(
        sNetID := ,
        hDBID := 1,
        cbCmdSize := SIZEOF(cmdSlc),
        pCmdAddr := ADR(cmdSlc),
        nStartIndex := 0,
        nRecordCount := 1,
        cbRecordArraySize := SIZEOF(lastCalibID),
        pDestAddr := ADR(lastCalibID),
        bExecute := bExecute,
        tTimeout := T#15S,
        bBusy => busy,
        bError => err,
        nErrID => errid,
        sSQLState => sqlstate,
        nRecords => recAnz
    );

    IF FB_SelectArray.bError THEN
        bInitSelectLastPumpCalibration := FALSE;
        GVL_Reports.bLoadBusy   := FALSE;
        GVL_Reports.bLoadDone   := FALSE;
        GVL_Reports.bLoadError  := TRUE;
        GVL_Reports.sLoadStatus := 'Error loading last pump calibration report';
        state := E_DB_QUERY_STATE.ERROR_STATE;

    ELSIF NOT FB_SelectArray.bBusy AND bInitSelectLastPumpCalibration THEN
        bInitSelectLastPumpCalibration := FALSE;

        IF recAnz > 0 AND lastCalibID[0] > 0 THEN
            GVL_Reports.sSelectedPrimaryID := INT_TO_STRING(lastCalibID[0]);
            DB_Query.state := E_DB_QUERY_STATE.SELECT_CALIB_REPORT_BY_ID;
        ELSE
            GVL_Reports.bLoadBusy   := FALSE;
            GVL_Reports.bLoadDone   := FALSE;
            GVL_Reports.bLoadError  := TRUE;
            GVL_Reports.sLoadStatus := 'No pump calibration report found';
            state := E_DB_QUERY_STATE.IDLE_STATE;
        END_IF

    ELSE
        state := E_DB_QUERY_STATE.SELECT_LAST_PUMP_CALIBRATION;
    END_IF

E_DB_QUERY_STATE.SELECT_SYSTEM_HISTORY_REPORT:

    GVL_Reports.bLoadBusy   := TRUE;
    GVL_Reports.bLoadDone   := FALSE;
    GVL_Reports.bLoadError  := FALSE;
    GVL_Reports.sLoadStatus := 'Loading system settings history report...';

    IF NOT bInitSelectSystemHistoryReport THEN
        bInitSelectSystemHistoryReport := TRUE;

        cmdSlc := GVL_DB.slctAllSys;
        bExecute := TRUE;
    ELSE
        bExecute := FALSE;
    END_IF

    FB_SelectArray(
        sNetID := ,
        hDBID := 1,
        cbCmdSize := SIZEOF(cmdSlc),
        pCmdAddr := ADR(cmdSlc),
        nStartIndex := 0,
        nRecordCount := 500,
        cbRecordArraySize := SIZEOF(GVL_Reports.aSystemHistory),
        pDestAddr := ADR(GVL_Reports.aSystemHistory),
        bExecute := bExecute,
        tTimeout := T#15S,
        bBusy => busy,
        bError => err,
        nErrID => errid,
        sSQLState => sqlstate,
        nRecords => recAnz
    );

    IF FB_SelectArray.bError THEN
        bInitSelectSystemHistoryReport := FALSE;
        GVL_Reports.bLoadBusy   := FALSE;
        GVL_Reports.bLoadDone   := FALSE;
        GVL_Reports.bLoadError  := TRUE;
        GVL_Reports.sLoadStatus := 'Error loading system settings history report';
        state := E_DB_QUERY_STATE.ERROR_STATE;

    ELSIF NOT FB_SelectArray.bBusy AND bInitSelectSystemHistoryReport THEN
        bInitSelectSystemHistoryReport := FALSE;
        GVL_Reports.bLoadBusy      := FALSE;
        GVL_Reports.bLoadDone      := TRUE;
        GVL_Reports.bLoadError     := FALSE;
        GVL_Reports.bPdfDataReady  := TRUE;
        GVL_Reports.bPdfConsumed   := FALSE;
        GVL_Reports.sLoadStatus    := 'System settings history report loaded';
        state := E_DB_QUERY_STATE.IDLE_STATE;

    ELSE
        state := E_DB_QUERY_STATE.SELECT_SYSTEM_HISTORY_REPORT;
    END_IF
	
E_DB_QUERY_STATE.SELECT_LINEAR_HISTORY_REPORT:

    GVL_Reports.bLoadBusy   := TRUE;
    GVL_Reports.bLoadDone   := FALSE;
    GVL_Reports.bLoadError  := FALSE;
    GVL_Reports.sLoadStatus := 'Loading linear pumps history report...';

    IF NOT bInitSelectLinearHistoryReport THEN
        bInitSelectLinearHistoryReport := TRUE;

        cmdSlc := GVL_DB.slctLinearHistoryReport;
        bExecute := TRUE;
    ELSE
        bExecute := FALSE;
    END_IF

    FB_SelectArray(
        sNetID := ,
        hDBID := 1,
        cbCmdSize := SIZEOF(cmdSlc),
        pCmdAddr := ADR(cmdSlc),
        nStartIndex := 0,
        nRecordCount := 200,
        cbRecordArraySize := SIZEOF(GVL_Reports.aLinearHistory),
        pDestAddr := ADR(GVL_Reports.aLinearHistory),
        bExecute := bExecute,
        tTimeout := T#15S,
        bBusy => busy,
        bError => err,
        nErrID => errid,
        sSQLState => sqlstate,
        nRecords => recAnz
    );

    IF FB_SelectArray.bError THEN
        bInitSelectLinearHistoryReport := FALSE;
        GVL_Reports.bLoadBusy   := FALSE;
        GVL_Reports.bLoadDone   := FALSE;
        GVL_Reports.bLoadError  := TRUE;
        GVL_Reports.sLoadStatus := 'Error loading linear pumps history report';
        state := E_DB_QUERY_STATE.ERROR_STATE;

    ELSIF NOT FB_SelectArray.bBusy AND bInitSelectLinearHistoryReport THEN
        bInitSelectLinearHistoryReport := FALSE;
        GVL_Reports.bLoadBusy      := FALSE;
        GVL_Reports.bLoadDone      := TRUE;
        GVL_Reports.bLoadError     := FALSE;
        GVL_Reports.bPdfDataReady  := TRUE;
        GVL_Reports.bPdfConsumed   := FALSE;
        GVL_Reports.sLoadStatus    := 'Linear pumps history report loaded';
        state := E_DB_QUERY_STATE.IDLE_STATE;

    ELSE
        state := E_DB_QUERY_STATE.SELECT_LINEAR_HISTORY_REPORT;
    END_IF
	
E_DB_QUERY_STATE.SELECT_COMPLETE_METHOD_REPORT:

    GVL_Reports.bLoadBusy   := TRUE;
    GVL_Reports.bLoadDone   := FALSE;
    GVL_Reports.bLoadError  := FALSE;
    GVL_Reports.sLoadStatus := 'Loading complete method history report...';

    IF NOT bInitSelectCompleteMethodReport THEN
        bInitSelectCompleteMethodReport := TRUE;
        bInitSelectCompleteMethodVolumes := FALSE;
        iCompleteMethodIndex := 1;

        Clear_CompleteMethodHeaderBuffer();
        Clear_CompleteMethodReportBuffer();

        cmdSlc := GVL_DB.slctAllMethodsForCompleteReport;
        bExecute := TRUE;
    ELSE
        bExecute := FALSE;
    END_IF

    FB_SelectArray(
        sNetID := ,
        hDBID := 1,
        cbCmdSize := SIZEOF(cmdSlc),
        pCmdAddr := ADR(cmdSlc),
        nStartIndex := 0,
        nRecordCount := 50,
        cbRecordArraySize := SIZEOF(GVL_Reports.aCompleteMethodHeader),
        pDestAddr := ADR(GVL_Reports.aCompleteMethodHeader),
        bExecute := bExecute,
        tTimeout := T#15S,
        bBusy => busy,
        bError => err,
        nErrID => errid,
        sSQLState => sqlstate,
        nRecords => recAnz
    );

    IF FB_SelectArray.bError THEN
        bInitSelectCompleteMethodReport := FALSE;
        GVL_Reports.bLoadBusy   := FALSE;
        GVL_Reports.bLoadDone   := FALSE;
        GVL_Reports.bLoadError  := TRUE;
        GVL_Reports.sLoadStatus := 'Error loading complete method history report';
        state := E_DB_QUERY_STATE.ERROR_STATE;

    ELSIF NOT FB_SelectArray.bBusy AND bInitSelectCompleteMethodReport THEN
        bInitSelectCompleteMethodReport := FALSE;

        IF recAnz > 0 THEN
            iCompleteMethodIndex := 1;
            state := E_DB_QUERY_STATE.SELECT_COMPLETE_METHOD_REPORT_VOLUMES;
        ELSE
            GVL_Reports.bLoadBusy   := FALSE;
            GVL_Reports.bLoadDone   := FALSE;
            GVL_Reports.bLoadError  := TRUE;
            GVL_Reports.sLoadStatus := 'No method history records found';
            state := E_DB_QUERY_STATE.IDLE_STATE;
        END_IF

    ELSE
        state := E_DB_QUERY_STATE.SELECT_COMPLETE_METHOD_REPORT;
    END_IF

E_DB_QUERY_STATE.SELECT_COMPLETE_METHOD_REPORT_VOLUMES:

    GVL_Reports.bLoadBusy   := TRUE;
    GVL_Reports.bLoadDone   := FALSE;
    GVL_Reports.bLoadError  := FALSE;
    GVL_Reports.sLoadStatus := 'Loading method volume data...';

    IF iCompleteMethodIndex > 50 OR GVL_Reports.aCompleteMethodHeader[iCompleteMethodIndex].methodID = 0 THEN
        GVL_Reports.bLoadBusy      := FALSE;
        GVL_Reports.bLoadDone      := TRUE;
        GVL_Reports.bLoadError     := FALSE;
        GVL_Reports.bPdfDataReady  := TRUE;
        GVL_Reports.bPdfConsumed   := FALSE;
        GVL_Reports.sLoadStatus    := 'Complete method history report loaded';
        state := E_DB_QUERY_STATE.IDLE_STATE;

    ELSE
        // Copy flat header into final struct
        GVL_Reports.aCompleteMethodReport[iCompleteMethodIndex].methodName := GVL_Reports.aCompleteMethodHeader[iCompleteMethodIndex].methodName;
        GVL_Reports.aCompleteMethodReport[iCompleteMethodIndex].methodRevision := GVL_Reports.aCompleteMethodHeader[iCompleteMethodIndex].methodRevision;
        GVL_Reports.aCompleteMethodReport[iCompleteMethodIndex].methodCreatedBy := GVL_Reports.aCompleteMethodHeader[iCompleteMethodIndex].methodCreatedBy;
        GVL_Reports.aCompleteMethodReport[iCompleteMethodIndex].methodCreatedOn := GVL_Reports.aCompleteMethodHeader[iCompleteMethodIndex].methodCreatedOn;
        GVL_Reports.aCompleteMethodReport[iCompleteMethodIndex].solvent_R1 := GVL_Reports.aCompleteMethodHeader[iCompleteMethodIndex].solvent_R1;
        GVL_Reports.aCompleteMethodReport[iCompleteMethodIndex].solvent_R2 := GVL_Reports.aCompleteMethodHeader[iCompleteMethodIndex].solvent_R2;
        GVL_Reports.aCompleteMethodReport[iCompleteMethodIndex].solvent_W1 := GVL_Reports.aCompleteMethodHeader[iCompleteMethodIndex].solvent_W1;
        GVL_Reports.aCompleteMethodReport[iCompleteMethodIndex].solvent_W2 := GVL_Reports.aCompleteMethodHeader[iCompleteMethodIndex].solvent_W2;
        GVL_Reports.aCompleteMethodReport[iCompleteMethodIndex].time_R1 := GVL_Reports.aCompleteMethodHeader[iCompleteMethodIndex].time_R1;
        GVL_Reports.aCompleteMethodReport[iCompleteMethodIndex].time_R2 := GVL_Reports.aCompleteMethodHeader[iCompleteMethodIndex].time_R2;
        GVL_Reports.aCompleteMethodReport[iCompleteMethodIndex].time_W1 := GVL_Reports.aCompleteMethodHeader[iCompleteMethodIndex].time_W1;
        GVL_Reports.aCompleteMethodReport[iCompleteMethodIndex].time_W2 := GVL_Reports.aCompleteMethodHeader[iCompleteMethodIndex].time_W2;
        GVL_Reports.aCompleteMethodReport[iCompleteMethodIndex].velocity_R1 := GVL_Reports.aCompleteMethodHeader[iCompleteMethodIndex].velocity_R1;
        GVL_Reports.aCompleteMethodReport[iCompleteMethodIndex].velocity_R2 := GVL_Reports.aCompleteMethodHeader[iCompleteMethodIndex].velocity_R2;
        GVL_Reports.aCompleteMethodReport[iCompleteMethodIndex].velocity_W1 := GVL_Reports.aCompleteMethodHeader[iCompleteMethodIndex].velocity_W1;
        GVL_Reports.aCompleteMethodReport[iCompleteMethodIndex].velocity_W2 := GVL_Reports.aCompleteMethodHeader[iCompleteMethodIndex].velocity_W2;
        GVL_Reports.aCompleteMethodReport[iCompleteMethodIndex].soakTime := GVL_Reports.aCompleteMethodHeader[iCompleteMethodIndex].soakTime;
        GVL_Reports.aCompleteMethodReport[iCompleteMethodIndex].agitate_1_Time := GVL_Reports.aCompleteMethodHeader[iCompleteMethodIndex].agitate_1_Time;
        GVL_Reports.aCompleteMethodReport[iCompleteMethodIndex].agitate_2_Time := GVL_Reports.aCompleteMethodHeader[iCompleteMethodIndex].agitate_2_Time;
        GVL_Reports.aCompleteMethodReport[iCompleteMethodIndex].vialsToFill := GVL_Reports.aCompleteMethodHeader[iCompleteMethodIndex].vialsToFill;
        GVL_Reports.aCompleteMethodReport[iCompleteMethodIndex].vialPrimeVol := GVL_Reports.aCompleteMethodHeader[iCompleteMethodIndex].vialPrimeVol;
        GVL_Reports.aCompleteMethodReport[iCompleteMethodIndex].vial_1_FillVol := GVL_Reports.aCompleteMethodHeader[iCompleteMethodIndex].vial_1_FillVol;
        GVL_Reports.aCompleteMethodReport[iCompleteMethodIndex].vial_2_4_FillVol := GVL_Reports.aCompleteMethodHeader[iCompleteMethodIndex].vial_2_4_FillVol;
        GVL_Reports.aCompleteMethodReport[iCompleteMethodIndex].airDryTime := GVL_Reports.aCompleteMethodHeader[iCompleteMethodIndex].airDryTime;
        GVL_Reports.aCompleteMethodReport[iCompleteMethodIndex].methodID := GVL_Reports.aCompleteMethodHeader[iCompleteMethodIndex].methodID;
        GVL_Reports.aCompleteMethodReport[iCompleteMethodIndex].methodStatus := GVL_Reports.aCompleteMethodHeader[iCompleteMethodIndex].methodStatus;

        sCompleteMethodID := INT_TO_STRING(GVL_Reports.aCompleteMethodHeader[iCompleteMethodIndex].methodID);

        IF NOT bInitSelectCompleteMethodVolumes THEN
            bInitSelectCompleteMethodVolumes := TRUE;

            selectRecipeVolumeByID(start := TRUE, methodID := sCompleteMethodID);
            bExecute := TRUE;
        ELSE
            bExecute := FALSE;
        END_IF

        FB_SelectArray(
            sNetID := ,
            hDBID := 1,
            cbCmdSize := SIZEOF(cmdSlc),
            pCmdAddr := ADR(cmdSlc),
            nStartIndex := 0,
            nRecordCount := 10,
            cbRecordArraySize := SIZEOF(GVL_Reports.aCompleteMethodReport[iCompleteMethodIndex].volumeData),
            pDestAddr := ADR(GVL_Reports.aCompleteMethodReport[iCompleteMethodIndex].volumeData),
            bExecute := bExecute,
            tTimeout := T#15S,
            bBusy => busy,
            bError => err,
            nErrID => errid,
            sSQLState => sqlstate,
            nRecords => recAnz
        );

        IF FB_SelectArray.bError THEN
            bInitSelectCompleteMethodVolumes := FALSE;
            GVL_Reports.bLoadBusy   := FALSE;
            GVL_Reports.bLoadDone   := FALSE;
            GVL_Reports.bLoadError  := TRUE;
            GVL_Reports.sLoadStatus := 'Error loading method volume data';
            state := E_DB_QUERY_STATE.ERROR_STATE;

        ELSIF NOT FB_SelectArray.bBusy AND bInitSelectCompleteMethodVolumes THEN
            bInitSelectCompleteMethodVolumes := FALSE;
            iCompleteMethodIndex := iCompleteMethodIndex + 1;
            state := E_DB_QUERY_STATE.SELECT_COMPLETE_METHOD_REPORT_VOLUMES;

        ELSE
            state := E_DB_QUERY_STATE.SELECT_COMPLETE_METHOD_REPORT_VOLUMES;
        END_IF
    END_IF

E_DB_QUERY_STATE.INSERT_USER_MGMT_HISTORY:

    cmdIn := GVL_DB.isrtUserMgmtHistory;

    insertUserMgmtHistory(start := TRUE);

    GVL_HMI.stUserMgmtHistoryEvent.bBusy := TRUE;
    GVL_HMI.stUserMgmtHistoryEvent.bDone := FALSE;
    GVL_HMI.stUserMgmtHistoryEvent.bError := FALSE;
    GVL_HMI.stUserMgmtHistoryEvent.sErrorText := '';

    FB_Insert(
        sNetID := ,
        hDBID := 1,
        cbCmdSize := SIZEOF(cmdIn),
        pCmdAddr := ADR(cmdIn),
        bExecute := TRUE,
        tTimeout := T#15S,
        bBusy => busy,
        bError => err,
        nErrID => errid,
        sSQLState => sqlstate
    );

    IF FB_Insert.bError THEN

		GVL_HMI.stUserMgmtHistoryEvent.bExecute := FALSE;
		GVL_HMI.stUserMgmtHistoryEvent.bBusy := FALSE;
		GVL_HMI.stUserMgmtHistoryEvent.bDone := FALSE;
		GVL_HMI.stUserMgmtHistoryEvent.bError := TRUE;
		GVL_HMI.stUserMgmtHistoryEvent.sErrorText := CONCAT('DB insert error. SQLState: ', sqlstate.sSQLState);
	
		state := E_DB_QUERY_STATE.ERROR_STATE;
		bExecuteIn := FALSE;
	
	ELSIF NOT FB_Insert.bBusy THEN
	
		GVL_HMI.stUserMgmtHistoryEvent.bExecute := FALSE;
		GVL_HMI.stUserMgmtHistoryEvent.bBusy := FALSE;
		GVL_HMI.stUserMgmtHistoryEvent.bDone := TRUE;
		GVL_HMI.stUserMgmtHistoryEvent.bError := FALSE;
		GVL_HMI.stUserMgmtHistoryEvent.sErrorText := '';
	
		state := E_DB_QUERY_STATE.IDLE_STATE;
		bExecuteIn := FALSE;
	
	ELSE
	
		state := E_DB_QUERY_STATE.INSERT_USER_MGMT_HISTORY;
		bExecuteIn := FALSE;
	
	END_IF
	
E_DB_QUERY_STATE.ERROR_STATE:

	bExecute:= FALSE;
	status:= 'SQL Error!';
	state:= E_DB_QUERY_STATE.IDLE_STATE;
		
END_CASE

METHOD Clear_CompleteMethodHeaderBuffer : BOOL
VAR_INPUT
END_VAR
VAR
    i : INT;
END_VAR
FOR i := 1 TO 50 DO
    GVL_Reports.aCompleteMethodHeader[i].methodName := '';
    GVL_Reports.aCompleteMethodHeader[i].methodRevision := '';
    GVL_Reports.aCompleteMethodHeader[i].methodCreatedBy := '';
    GVL_Reports.aCompleteMethodHeader[i].methodCreatedOn := '';
    GVL_Reports.aCompleteMethodHeader[i].solvent_R1 := '';
    GVL_Reports.aCompleteMethodHeader[i].solvent_R2 := '';
    GVL_Reports.aCompleteMethodHeader[i].solvent_W1 := '';
    GVL_Reports.aCompleteMethodHeader[i].solvent_W2 := '';
    GVL_Reports.aCompleteMethodHeader[i].time_R1 := '';
    GVL_Reports.aCompleteMethodHeader[i].time_R2 := '';
    GVL_Reports.aCompleteMethodHeader[i].time_W1 := '';
    GVL_Reports.aCompleteMethodHeader[i].time_W2 := '';
    GVL_Reports.aCompleteMethodHeader[i].velocity_R1 := '';
    GVL_Reports.aCompleteMethodHeader[i].velocity_R2 := '';
    GVL_Reports.aCompleteMethodHeader[i].velocity_W1 := '';
    GVL_Reports.aCompleteMethodHeader[i].velocity_W2 := '';
    GVL_Reports.aCompleteMethodHeader[i].soakTime := '';
    GVL_Reports.aCompleteMethodHeader[i].agitate_1_Time := '';
    GVL_Reports.aCompleteMethodHeader[i].agitate_2_Time := '';
    GVL_Reports.aCompleteMethodHeader[i].vialsToFill := '';
    GVL_Reports.aCompleteMethodHeader[i].vialPrimeVol := '';
    GVL_Reports.aCompleteMethodHeader[i].vial_1_FillVol := '';
    GVL_Reports.aCompleteMethodHeader[i].vial_2_4_FillVol := '';
    GVL_Reports.aCompleteMethodHeader[i].airDryTime := '';
    GVL_Reports.aCompleteMethodHeader[i].methodID := 0;
    GVL_Reports.aCompleteMethodHeader[i].methodStatus := '';
END_FOR
END_METHOD

METHOD Clear_CompleteMethodReportBuffer : BOOL
VAR
	i, j : INT;
END_VAR
FOR i := 1 TO 50 DO
    GVL_Reports.aCompleteMethodReport[i].methodName := '';
    GVL_Reports.aCompleteMethodReport[i].methodRevision := '';
    GVL_Reports.aCompleteMethodReport[i].methodCreatedBy := '';
    GVL_Reports.aCompleteMethodReport[i].methodCreatedOn := '';
    GVL_Reports.aCompleteMethodReport[i].solvent_R1 := '';
    GVL_Reports.aCompleteMethodReport[i].solvent_R2 := '';
    GVL_Reports.aCompleteMethodReport[i].solvent_W1 := '';
    GVL_Reports.aCompleteMethodReport[i].solvent_W2 := '';
    GVL_Reports.aCompleteMethodReport[i].time_R1 := '';
    GVL_Reports.aCompleteMethodReport[i].time_R2 := '';
    GVL_Reports.aCompleteMethodReport[i].time_W1 := '';
    GVL_Reports.aCompleteMethodReport[i].time_W2 := '';
    GVL_Reports.aCompleteMethodReport[i].velocity_R1 := '';
    GVL_Reports.aCompleteMethodReport[i].velocity_R2 := '';
    GVL_Reports.aCompleteMethodReport[i].velocity_W1 := '';
    GVL_Reports.aCompleteMethodReport[i].velocity_W2 := '';
    GVL_Reports.aCompleteMethodReport[i].soakTime := '';
    GVL_Reports.aCompleteMethodReport[i].agitate_1_Time := '';
    GVL_Reports.aCompleteMethodReport[i].agitate_2_Time := '';
    GVL_Reports.aCompleteMethodReport[i].vialsToFill := '';
    GVL_Reports.aCompleteMethodReport[i].vialPrimeVol := '';
    GVL_Reports.aCompleteMethodReport[i].vial_1_FillVol := '';
    GVL_Reports.aCompleteMethodReport[i].vial_2_4_FillVol := '';
    GVL_Reports.aCompleteMethodReport[i].airDryTime := '';
    GVL_Reports.aCompleteMethodReport[i].methodID := 0;
    GVL_Reports.aCompleteMethodReport[i].methodStatus := '';

    FOR j := 1 TO 10 DO
        GVL_Reports.aCompleteMethodReport[i].volumeData[j].VD_ID := 0;
        GVL_Reports.aCompleteMethodReport[i].volumeData[j].pump := '';
        GVL_Reports.aCompleteMethodReport[i].volumeData[j].stage := '';
        GVL_Reports.aCompleteMethodReport[i].volumeData[j].rinse1 := '';
        GVL_Reports.aCompleteMethodReport[i].volumeData[j].rinse2 := '';
        GVL_Reports.aCompleteMethodReport[i].volumeData[j].wash1 := '';
        GVL_Reports.aCompleteMethodReport[i].volumeData[j].wash2 := '';
        GVL_Reports.aCompleteMethodReport[i].volumeData[j].methodID := 0;
    END_FOR
END_FOR
END_METHOD

METHOD Clear_LinearReportBuffer : BOOL
VAR_INPUT
END_VAR
GVL_Reports.stLinearReport.ID_Linear := 0;
GVL_Reports.stLinearReport.pump1 := '';
GVL_Reports.stLinearReport.pump2 := '';
GVL_Reports.stLinearReport.pump3 := '';
GVL_Reports.stLinearReport.pump4 := '';
GVL_Reports.stLinearReport.pump5 := '';
GVL_Reports.stLinearReport.pump6 := '';
GVL_Reports.stLinearReport.pump7 := '';
GVL_Reports.stLinearReport.pump8 := '';
GVL_Reports.stLinearReport.pump9 := '';
GVL_Reports.stLinearReport.pump10 := '';
GVL_Reports.stLinearReport.changedBy := '';
GVL_Reports.stLinearReport.changedOn := '';
END_METHOD

METHOD Clear_MethodReportBuffers : BOOL
VAR
	i : INT;
END_VAR
GVL_Reports.stMethodHeader.methodName := '';
GVL_Reports.stMethodHeader.methodRevision := '';
GVL_Reports.stMethodHeader.methodCreatedBy := '';
GVL_Reports.stMethodHeader.methodCreatedOn := '';
GVL_Reports.stMethodHeader.solvent_R1 := '';
GVL_Reports.stMethodHeader.solvent_R2 := '';
GVL_Reports.stMethodHeader.solvent_W1 := '';
GVL_Reports.stMethodHeader.solvent_W2 := '';
GVL_Reports.stMethodHeader.time_R1 := '';
GVL_Reports.stMethodHeader.time_R2 := '';
GVL_Reports.stMethodHeader.time_W1 := '';
GVL_Reports.stMethodHeader.time_W2 := '';
GVL_Reports.stMethodHeader.velocity_R1 := '';
GVL_Reports.stMethodHeader.velocity_R2 := '';
GVL_Reports.stMethodHeader.velocity_W1 := '';
GVL_Reports.stMethodHeader.velocity_W2 := '';
GVL_Reports.stMethodHeader.soakTime := '';
GVL_Reports.stMethodHeader.agitate_1_Time := '';
GVL_Reports.stMethodHeader.agitate_2_Time := '';
GVL_Reports.stMethodHeader.vialsToFill := '';
GVL_Reports.stMethodHeader.vialPrimeVol := '';
GVL_Reports.stMethodHeader.vial_1_FillVol := '';
GVL_Reports.stMethodHeader.vial_2_4_FillVol := '';
GVL_Reports.stMethodHeader.airDryTime := '';
GVL_Reports.stMethodHeader.methodID := 0;
GVL_Reports.stMethodHeader.methodStatus := '';

FOR i := 1 TO 10 DO
    GVL_Reports.aMethodVolumeData[i].pump := '';
    GVL_Reports.aMethodVolumeData[i].stage := '';
    GVL_Reports.aMethodVolumeData[i].rinse1 := '';
    GVL_Reports.aMethodVolumeData[i].rinse2 := '';
    GVL_Reports.aMethodVolumeData[i].wash1 := '';
    GVL_Reports.aMethodVolumeData[i].wash2 := '';
END_FOR
END_METHOD

METHOD Clear_PostRunBuffers : BOOL
VAR
	i : INT;
END_VAR
GVL_Reports.stRunHeader.runNo := 0;
GVL_Reports.stRunHeader.analyst := '';
GVL_Reports.stRunHeader.comment := '';
GVL_Reports.stRunHeader.softwareVersion := '';
GVL_Reports.stRunHeader.sysMasterRevision := '';
GVL_Reports.stRunHeader.sysSettingsRevision := '';
GVL_Reports.stRunHeader.meterVelocity := '';
GVL_Reports.stRunHeader.runVelocity := '';
GVL_Reports.stRunHeader.emptyTubesFactor := '';
GVL_Reports.stRunHeader.fillTubesFactor := '';
GVL_Reports.stRunHeader.solvent1NameRevision := '';
GVL_Reports.stRunHeader.solvent2NameRevision := '';
GVL_Reports.stRunHeader.solvent3NameRevision := '';
GVL_Reports.stRunHeader.solvent4NameRevision := '';
GVL_Reports.stRunHeader.timeEventStarted := '';
GVL_Reports.stRunHeader.timeEventCompleted := '';
GVL_Reports.stRunHeader.methodID := 0;
GVL_Reports.stRunHeader.CalibrationNo := 0;

GVL_Reports.stRunMethodHeader.methodName := '';
GVL_Reports.stRunMethodHeader.methodRevision := '';
GVL_Reports.stRunMethodHeader.methodCreatedBy := '';
GVL_Reports.stRunMethodHeader.methodCreatedOn := '';
GVL_Reports.stRunMethodHeader.solvent_R1 := '';
GVL_Reports.stRunMethodHeader.solvent_R2 := '';
GVL_Reports.stRunMethodHeader.solvent_W1 := '';
GVL_Reports.stRunMethodHeader.solvent_W2 := '';
GVL_Reports.stRunMethodHeader.time_R1 := '';
GVL_Reports.stRunMethodHeader.time_R2 := '';
GVL_Reports.stRunMethodHeader.time_W1 := '';
GVL_Reports.stRunMethodHeader.time_W2 := '';
GVL_Reports.stRunMethodHeader.velocity_R1 := '';
GVL_Reports.stRunMethodHeader.velocity_R2 := '';
GVL_Reports.stRunMethodHeader.velocity_W1 := '';
GVL_Reports.stRunMethodHeader.velocity_W2 := '';
GVL_Reports.stRunMethodHeader.soakTime := '';
GVL_Reports.stRunMethodHeader.agitate_1_Time := '';
GVL_Reports.stRunMethodHeader.agitate_2_Time := '';
GVL_Reports.stRunMethodHeader.vialsToFill := '';
GVL_Reports.stRunMethodHeader.vialPrimeVol := '';
GVL_Reports.stRunMethodHeader.vial_1_FillVol := '';
GVL_Reports.stRunMethodHeader.vial_2_4_FillVol := '';
GVL_Reports.stRunMethodHeader.airDryTime := '';
GVL_Reports.stRunMethodHeader.methodID := 0;
GVL_Reports.stRunMethodHeader.methodStatus := '';

FOR i := 1 TO 10 DO
    GVL_Reports.aRunVolumeData[i].VD_ID := 0;
    GVL_Reports.aRunVolumeData[i].pump := '';
    GVL_Reports.aRunVolumeData[i].stage := '';
    GVL_Reports.aRunVolumeData[i].rinse1 := '';
    GVL_Reports.aRunVolumeData[i].rinse2 := '';
    GVL_Reports.aRunVolumeData[i].wash1 := '';
    GVL_Reports.aRunVolumeData[i].wash2 := '';
    GVL_Reports.aRunVolumeData[i].methodID := 0;
END_FOR

sPostRunMethodID := '';
END_METHOD

METHOD Clear_PumpCalibReportBuffers : BOOL
VAR
	i : INT;
END_VAR
GVL_Reports.iPumpCalibNo           := 0;
GVL_Reports.sPumpCalibUserID       := '';
GVL_Reports.sPumpCalibDensity      := '';
GVL_Reports.sPumpCalibSolventNo    := '';
GVL_Reports.sPumpCalibSolventRev   := '';
GVL_Reports.sPumpCalibAllowFail    := '';
GVL_Reports.sPumpCalibReplicates   := '';
GVL_Reports.sPumpCalibCallInterval := '';
GVL_Reports.sPumpCalibSysRev       := '';

FOR i := 1 TO 100 DO
    GVL_Reports.aPumpCalibValues[i].CalibrationNo      := 0;
    GVL_Reports.aPumpCalibValues[i].dateTime           := '';
    GVL_Reports.aPumpCalibValues[i].pumpNo             := '';
    GVL_Reports.aPumpCalibValues[i].step               := '';
    GVL_Reports.aPumpCalibValues[i].tareWt             := '';
    GVL_Reports.aPumpCalibValues[i].grossWt            := '';
    GVL_Reports.aPumpCalibValues[i].netVolume          := '';
    GVL_Reports.aPumpCalibValues[i].netWt              := '';
    GVL_Reports.aPumpCalibValues[i].targetVolume       := '';
    GVL_Reports.aPumpCalibValues[i].differencePercent  := '';
    GVL_Reports.aPumpCalibValues[i].criteria           := '';
    GVL_Reports.aPumpCalibValues[i].pumpRevs           := '';
END_FOR

// Return flag
Clear_PumpCalibReportBuffers := TRUE;
END_METHOD

METHOD Clear_ReportSearchResult : BOOL
VAR
	i : INT;
END_VAR
FOR i := 1 TO 100 DO
    GVL_Reports.aReportSearchResult[i].ReportType  := '';
    GVL_Reports.aReportSearchResult[i].ReportID    := '';
    GVL_Reports.aReportSearchResult[i].CreatedOn   := '';
    GVL_Reports.aReportSearchResult[i].CreatedBy   := '';
    GVL_Reports.aReportSearchResult[i].Description := '';
    GVL_Reports.aReportSearchResult[i].sPrimaryKey := '';
END_FOR

GVL_Reports.uiReportSearchCount := 0;
GVL_Reports.sDateFromFilter  := '';
GVL_Reports.sQuickReportName := '';
GVL_Reports.sDateToFilter    := '';
GVL_Reports.sQuickReportName := '';
GVL_Reports.bUseDateFilter   := FALSE;

bInitSelectCalibReportList := FALSE;
bInitSelectSystemSettingsReportList := FALSE;

bInitSelectCalibReportByID 			  := FALSE;
bInitSelectCalibReportValuesByID	  := FALSE;
bInitSelectSystemSettingsReportList   := FALSE;
bInitSelectSystemSettingsByID         := FALSE;
bInitSelectCalibReportList			  := FALSE;
bInitSelectMethodReportList			  := FALSE;
bInitSelectMethodReportSearch		  := FALSE;
bInitSelectRunReportList			  := FALSE;
bInitSelectRecipeHeaderByID 		  := FALSE;
bInitSelectRecipeVolumeByID 		  := FALSE;
bInitSelectLinearByID 				  := FALSE;
bInitSelectPostRunByID 				  := FALSE;
bInitSelectPostRunMethodByID 		  := FALSE;
bInitSelectPostRunVolumeByMethodID 	  := FALSE;
bInitSelectLinearReportSearch 		  := FALSE;
bInitSelectLastLinearReport 		  := FALSE;
bInitSelectLastPostRunRun  			  := FALSE;
bInitSelectLastPumpCalibration  	  := FALSE;
bInitSelectSystemHistoryReport 		  := FALSE;
bInitSelectLinearHistoryReport 		  := FALSE;
bInitSelectCompleteMethodReport 	  := FALSE;
bInitSelectCompleteMethodVolumes 	  := FALSE;
iCompleteMethodIndex := 1;


GVL_Reports.sDateFromFilter := '';
GVL_Reports.sDateToFilter   := '';
GVL_Reports.bUseDateFilter  := FALSE;
GVL_Reports.bClearDateFilters := FALSE;

cmdSlc := '';
recAnz := 0;
bExecute := FALSE;
busy := FALSE;
err := FALSE;
errid := 0;
//sqlstate := '';

// Return flag
Clear_ReportSearchResult := TRUE;
END_METHOD

METHOD Clear_SystemSettingsReportBuffer : BOOL
VAR_INPUT
END_VAR
GVL_Reports.stSelectedSystemSettings.sGenSealAndPump            := '';
GVL_Reports.stSelectedSystemSettings.sCalAcceptanceCriteria     := '';
GVL_Reports.stSelectedSystemSettings.sCalAllowableFail          := '';
GVL_Reports.stSelectedSystemSettings.sCalReplicates             := '';
GVL_Reports.stSelectedSystemSettings.sCalPumpCallIntervalDays   := '';
GVL_Reports.stSelectedSystemSettings.sCalCloseAppOnCompletion   := '';
GVL_Reports.stSelectedSystemSettings.sAirDryTimeOnCompletion    := '';
GVL_Reports.stSelectedSystemSettings.sLktAllowableLeakTestFail  := '';
GVL_Reports.stSelectedSystemSettings.sLktLeakTestBuildUpTime    := '';
GVL_Reports.stSelectedSystemSettings.sLktLeakTestHoldTime       := '';
GVL_Reports.stSelectedSystemSettings.sLktLeakTestPressure       := '';
GVL_Reports.stSelectedSystemSettings.sMecPlatesClosedPosition   := '';
GVL_Reports.stSelectedSystemSettings.sMecPlatesDryPosition      := '';
GVL_Reports.stSelectedSystemSettings.sMecPlatesVelocity         := '';
GVL_Reports.stSelectedSystemSettings.sMecMaxCurrentFastDown     := '';
GVL_Reports.stSelectedSystemSettings.sMecMaxCurrentSlowDown     := '';
GVL_Reports.stSelectedSystemSettings.sMecMaxCurrentSlowUp       := '';
GVL_Reports.stSelectedSystemSettings.sPmpMeterVelocity          := '';
GVL_Reports.stSelectedSystemSettings.sPmpRunVelocity            := '';
GVL_Reports.stSelectedSystemSettings.sPmpEmptyFactor            := '';
GVL_Reports.stSelectedSystemSettings.sPmpFillSolventTubesFactor := '';
GVL_Reports.stSelectedSystemSettings.sSmpAboveCalibration       := '';
GVL_Reports.stSelectedSystemSettings.sSmpVialSetSpacing         := '';
GVL_Reports.stSelectedSystemSettings.sSmpIntoResBottom          := '';
GVL_Reports.stSelectedSystemSettings.sSmpIntoResDispense        := '';
GVL_Reports.stSelectedSystemSettings.sSmpIntoResWeigh           := '';
GVL_Reports.stSelectedSystemSettings.sSmpIntoVials              := '';
GVL_Reports.stSelectedSystemSettings.sSmpIntoWaste              := '';
GVL_Reports.stSelectedSystemSettings.sSecDisplayManualControl   := '';
GVL_Reports.stSelectedSystemSettings.sSecCheckLogonEachRun      := '';
GVL_Reports.stSelectedSystemSettings.sCreatedBy                 := '';
GVL_Reports.stSelectedSystemSettings.sCreatedDate               := '';
GVL_Reports.stSelectedSystemSettings.sSysRevisionNo             := '';
END_METHOD

METHOD copyPumpCalibHeaderToReports : BOOL
VAR_INPUT
END_VAR
GVL_Reports.iPumpCalibNo           := aPumpCalibHeader[1].CalibrationNo;
GVL_Reports.sPumpCalibUserID       := aPumpCalibHeader[1].userID;
GVL_Reports.sPumpCalibDensity      := aPumpCalibHeader[1].density;
GVL_Reports.sPumpCalibSolventNo    := aPumpCalibHeader[1].solventNo;
GVL_Reports.sPumpCalibSolventRev   := aPumpCalibHeader[1].solventRevision;
GVL_Reports.sPumpCalibAllowFail    := aPumpCalibHeader[1].allowableFail;
GVL_Reports.sPumpCalibReplicates   := aPumpCalibHeader[1].replicates;
GVL_Reports.sPumpCalibCallInterval := aPumpCalibHeader[1].callInterval;
GVL_Reports.sPumpCalibSysRev       := INT_TO_STRING(aPumpCalibHeader[1].sysRevisionNo);
END_METHOD

METHOD CopySelectedCalibHeaderToLegacy : BOOL
VAR_INPUT
END_VAR
GVL_Reports.iPumpCalibNo           := STRING_TO_INT(GVL_Reports.stSelectedCalibReportHeader.sCalibrationNo);
GVL_Reports.sPumpCalibUserID       := GVL_Reports.stSelectedCalibReportHeader.sUserId;
GVL_Reports.sPumpCalibDensity      := GVL_Reports.stSelectedCalibReportHeader.sDensity;
GVL_Reports.sPumpCalibSolventNo    := GVL_Reports.stSelectedCalibReportHeader.sSolventNo;
GVL_Reports.sPumpCalibSolventRev   := GVL_Reports.stSelectedCalibReportHeader.sSolventRevision;
GVL_Reports.sPumpCalibSysRev       := GVL_Reports.stSelectedCalibReportHeader.sSysRevisionNo;
GVL_Reports.sPumpCalibAllowFail    := GVL_Reports.stSelectedCalibReportHeader.sAllowableFail;
GVL_Reports.sPumpCalibReplicates   := GVL_Reports.stSelectedCalibReportHeader.sReplicates;
GVL_Reports.sPumpCalibCallInterval := GVL_Reports.stSelectedCalibReportHeader.sCallInterval;
END_METHOD

METHOD CopySelectedCalibLinesToLegacy : BOOL
VAR
	 i : INT;
END_VAR
FOR i := 1 TO 100 DO
    GVL_Reports.aPumpCalibValues[i].dateTime          := '';
    GVL_Reports.aPumpCalibValues[i].pumpNo            := '';
    GVL_Reports.aPumpCalibValues[i].step              := '';
    GVL_Reports.aPumpCalibValues[i].tareWt            := '';
    GVL_Reports.aPumpCalibValues[i].grossWt           := '';
    GVL_Reports.aPumpCalibValues[i].netWt             := '';
    GVL_Reports.aPumpCalibValues[i].netVolume         := '';
    GVL_Reports.aPumpCalibValues[i].targetVolume      := '';
    GVL_Reports.aPumpCalibValues[i].differencePercent := '';
    GVL_Reports.aPumpCalibValues[i].criteria          := '';
    GVL_Reports.aPumpCalibValues[i].pumpRevs          := '';
END_FOR

FOR i := 1 TO 100 DO
    IF i <= 300 THEN
        GVL_Reports.aPumpCalibValues[i].dateTime          := GVL_Reports.aSelectedCalibReportLines[i].sDateTime;
        GVL_Reports.aPumpCalibValues[i].pumpNo            := GVL_Reports.aSelectedCalibReportLines[i].sPumpNo;
        GVL_Reports.aPumpCalibValues[i].step              := GVL_Reports.aSelectedCalibReportLines[i].sStep;
        GVL_Reports.aPumpCalibValues[i].tareWt            := GVL_Reports.aSelectedCalibReportLines[i].sTareWt;
        GVL_Reports.aPumpCalibValues[i].grossWt           := GVL_Reports.aSelectedCalibReportLines[i].sGrossWt;
        GVL_Reports.aPumpCalibValues[i].netWt             := GVL_Reports.aSelectedCalibReportLines[i].sNetWt;
        GVL_Reports.aPumpCalibValues[i].netVolume         := GVL_Reports.aSelectedCalibReportLines[i].sNetVolume;
        GVL_Reports.aPumpCalibValues[i].targetVolume      := GVL_Reports.aSelectedCalibReportLines[i].sTargetVolume;
        GVL_Reports.aPumpCalibValues[i].differencePercent := GVL_Reports.aSelectedCalibReportLines[i].sDifferencePercent;
        GVL_Reports.aPumpCalibValues[i].criteria          := GVL_Reports.aSelectedCalibReportLines[i].sCriteria;
        GVL_Reports.aPumpCalibValues[i].pumpRevs          := GVL_Reports.aSelectedCalibReportLines[i].sPumpRevs;
    END_IF
END_FOR
END_METHOD

METHOD deleteCalibHead : BOOL
VAR_INPUT
	start : BOOL;
END_VAR
VAR
	sCalibNo : STRING;
END_VAR
// Builds the DELETE command that removes an orphaned CALIBRATION_HEAD row.
// Called from E_DB_QUERY_STATE.DELETE_CALIBRATION_HEAD when calibration
// was aborted before any measurement row was inserted into [CALIBRATION].
sCalibNo := INT_TO_STRING(GVL_DB.stParameter_PCR.CalibrationNo);

IF start THEN
    FindAndReplace(
        pSrcString    := ADR(cmdIn),
        pDeleteString := ADR('#1#'),
        pInsertString := ADR(sCalibNo),
        pDstString    := ADR(cmdIn),
        nDstSize      := SIZEOF(cmdIn)
    );
END_IF
END_METHOD

METHOD Fill_Calibration_Data : BOOL
VAR_INPUT
END_VAR
FOR i:=1 TO 100 BY 1 DO 
GVL_DB.astData_PCR[i].CalibrationNo			:= 0;
GVL_DB.astData_PCR[i].criteria				:= '';
GVL_DB.astData_PCR[i].dateTime				:= '';
GVL_DB.astData_PCR[i].differencePercent		:= '';
GVL_DB.astData_PCR[i].grossWt				:= '';
GVL_DB.astData_PCR[i].netVolume				:= '';
GVL_DB.astData_PCR[i].netWt					:= '';
GVL_DB.astData_PCR[i].pumpNo				:= '';
GVL_DB.astData_PCR[i].pumpRevs				:= '';
GVL_DB.astData_PCR[i].step					:= '';
GVL_DB.astData_PCR[i].tareWt				:= '';
GVL_DB.astData_PCR[i].targetVolume			:= '';
END_FOR

FOR i:=1 TO 100 BY 1 DO 
GVL_DB.astData_PCR[i].CalibrationNo			:= GVL_DB.stParameter_PCR.CalibrationNo;
GVL_DB.astData_PCR[i].criteria				:= REAL_TO_STRING(GVL_Calibration.stPumpCalibrationData[i].rCriteria);
GVL_DB.astData_PCR[i].dateTime				:= GVL_Calibration.stPumpCalibrationData[i].dDateTime;
GVL_DB.astData_PCR[i].differencePercent		:= LREAL_TO_STRING(GVL_Calibration.stPumpCalibrationData[i].rDifferencePercent);
GVL_DB.astData_PCR[i].grossWt				:= LREAL_TO_STRING(GVL_Calibration.stPumpCalibrationData[i].rGrossWeigth);
GVL_DB.astData_PCR[i].netVolume				:= LREAL_TO_STRING(GVL_Calibration.stPumpCalibrationData[i].rNetVolume);
GVL_DB.astData_PCR[i].netWt					:= LREAL_TO_STRING(GVL_Calibration.stPumpCalibrationData[i].rNetWeigth);
GVL_DB.astData_PCR[i].pumpNo				:= USINT_TO_STRING(GVL_Calibration.stPumpCalibrationData[i].iPumpNumber);
GVL_DB.astData_PCR[i].pumpRevs				:= UINT_TO_STRING(GVL_Calibration.stPumpCalibrationData[i].iPumpRevs);
GVL_DB.astData_PCR[i].step					:= GVL_Calibration.stPumpCalibrationData[i].sStep;
GVL_DB.astData_PCR[i].tareWt				:= LREAL_TO_STRING(GVL_Calibration.stPumpCalibrationData[i].rTareWeigth);
GVL_DB.astData_PCR[i].targetVolume			:= LREAL_TO_STRING(GVL_Calibration.stPumpCalibrationData[i].rTargetVolume);
END_FOR
END_METHOD

METHOD Fill_Method_Data : BOOL
VAR_INPUT
END_VAR

VAR
	j: INT;
END_VAR

GVL_Recipe.stCurrentRecipe.stOtherParams.tAgitate1Time := DINT_TO_TIME(STRING_TO_DINT(GVL_DB.stParameter_MR.agitate_1_Time)*1000);
GVL_Recipe.stCurrentRecipe.stOtherParams.tAgitate2Time := DINT_TO_TIME(STRING_TO_DINT(GVL_DB.stParameter_MR.agitate_2_Time)*1000);
GVL_Recipe.stCurrentRecipe.stOtherParams.tAirDryTime := DINT_TO_TIME(STRING_TO_DINT(GVL_DB.stParameter_MR.airDryTime)*1000);
GVL_Recipe.stCurrentRecipe.stInfo.sCreatedBy := GVL_DB.stParameter_MR.methodCreatedBy;
//GVL_Recipe.stCurrentRecipe.stInfo.dCreationDate := GVL_DB.stParameter_MR.methodCreatedOn;
GVL_Recipe.stCurrentRecipe.stInfo.sMethodName := GVL_DB.stParameter_MR.methodName;
GVL_Recipe.stCurrentRecipe.stInfo.iRevision := STRING_TO_INT(GVL_DB.stParameter_MR.methodRevision);
GVL_Recipe.stCurrentRecipe.stOtherParams.tSoakTime := DINT_TO_TIME(STRING_TO_DINT(GVL_DB.stParameter_MR.soakTime)*1000);
GVL_Recipe.stCurrentRecipe.stSolventsTimes.aSolventN[1] := STRING_TO_USINT(GVL_DB.stParameter_MR.solvent_R1);
GVL_Recipe.stCurrentRecipe.stSolventsTimes.aSolventN[2] := STRING_TO_USINT(GVL_DB.stParameter_MR.solvent_R2);
GVL_Recipe.stCurrentRecipe.stSolventsTimes.aSolventN[3] := STRING_TO_USINT(GVL_DB.stParameter_MR.solvent_W1);
GVL_Recipe.stCurrentRecipe.stSolventsTimes.aSolventN[4] := STRING_TO_USINT(GVL_DB.stParameter_MR.solvent_W2);
GVL_Recipe.stCurrentRecipe.stSolventsTimes.aTime[1] := DINT_TO_TIME(STRING_TO_DINT(GVL_DB.stParameter_MR.time_R1)*1000);
GVL_Recipe.stCurrentRecipe.stSolventsTimes.aTime[2] := DINT_TO_TIME(STRING_TO_DINT(GVL_DB.stParameter_MR.time_R2)*1000);
GVL_Recipe.stCurrentRecipe.stSolventsTimes.aTime[3] := DINT_TO_TIME(STRING_TO_DINT(GVL_DB.stParameter_MR.time_W1)*1000);
GVL_Recipe.stCurrentRecipe.stSolventsTimes.aTime[4] := DINT_TO_TIME(STRING_TO_DINT(GVL_DB.stParameter_MR.time_W2)*1000);
GVL_Recipe.stCurrentRecipe.stSolventsTimes.aVelocity[1] := STRING_TO_INT(GVL_DB.stParameter_MR.velocity_R1);
GVL_Recipe.stCurrentRecipe.stSolventsTimes.aVelocity[2] := STRING_TO_INT(GVL_DB.stParameter_MR.velocity_R2);
GVL_Recipe.stCurrentRecipe.stSolventsTimes.aVelocity[3] := STRING_TO_INT(GVL_DB.stParameter_MR.velocity_W1);
GVL_Recipe.stCurrentRecipe.stSolventsTimes.aVelocity[4] := STRING_TO_INT(GVL_DB.stParameter_MR.velocity_W2);
GVL_Recipe.stCurrentRecipe.stOtherParams.rVial1FillVol := STRING_TO_REAL(GVL_DB.stParameter_MR.vial_1_FillVol);
GVL_Recipe.stCurrentRecipe.stOtherParams.rVials2_4FillVol := STRING_TO_REAL(GVL_DB.stParameter_MR.vial_2_4_FillVol);
GVL_Recipe.stCurrentRecipe.stOtherParams.rVialPrimeVol := STRING_TO_REAL(GVL_DB.stParameter_MR.vialPrimeVol);
GVL_Recipe.stCurrentRecipe.stOtherParams.iVialsToFill := STRING_TO_USINT(GVL_DB.stParameter_MR.vialsToFill);

GVL_Recipe.stCurrentRecipe.stVolumes.aT_IC_Volume[1] := STRING_TO_REAL(GVL_DB.astVolData[1].rinse1);
GVL_Recipe.stCurrentRecipe.stVolumes.aT_IC_Volume[2] := STRING_TO_REAL(GVL_DB.astVolData[1].rinse2);
GVL_Recipe.stCurrentRecipe.stVolumes.aT_IC_Volume[3] := STRING_TO_REAL(GVL_DB.astVolData[1].wash1);
GVL_Recipe.stCurrentRecipe.stVolumes.aT_IC_Volume[4] := STRING_TO_REAL(GVL_DB.astVolData[1].wash2);
GVL_Recipe.stCurrentRecipe.stVolumes.aS0_Volume[1] := STRING_TO_REAL(GVL_DB.astVolData[2].rinse1);
GVL_Recipe.stCurrentRecipe.stVolumes.aS0_Volume[2] := STRING_TO_REAL(GVL_DB.astVolData[2].rinse2);
GVL_Recipe.stCurrentRecipe.stVolumes.aS0_Volume[3] := STRING_TO_REAL(GVL_DB.astVolData[2].wash1);
GVL_Recipe.stCurrentRecipe.stVolumes.aS0_Volume[4] := STRING_TO_REAL(GVL_DB.astVolData[2].wash2);
GVL_Recipe.stCurrentRecipe.stVolumes.aS1_Volume[1] := STRING_TO_REAL(GVL_DB.astVolData[3].rinse1);
GVL_Recipe.stCurrentRecipe.stVolumes.aS1_Volume[2] := STRING_TO_REAL(GVL_DB.astVolData[3].rinse2);
GVL_Recipe.stCurrentRecipe.stVolumes.aS1_Volume[3] := STRING_TO_REAL(GVL_DB.astVolData[3].wash1);
GVL_Recipe.stCurrentRecipe.stVolumes.aS1_Volume[4] := STRING_TO_REAL(GVL_DB.astVolData[3].wash2);
GVL_Recipe.stCurrentRecipe.stVolumes.aS2_Volume[1] := STRING_TO_REAL(GVL_DB.astVolData[4].rinse1);
GVL_Recipe.stCurrentRecipe.stVolumes.aS2_Volume[2] := STRING_TO_REAL(GVL_DB.astVolData[4].rinse2);
GVL_Recipe.stCurrentRecipe.stVolumes.aS2_Volume[3] := STRING_TO_REAL(GVL_DB.astVolData[4].wash1);
GVL_Recipe.stCurrentRecipe.stVolumes.aS2_Volume[4] := STRING_TO_REAL(GVL_DB.astVolData[4].wash2);
GVL_Recipe.stCurrentRecipe.stVolumes.aS3_Volume[1] := STRING_TO_REAL(GVL_DB.astVolData[5].rinse1);
GVL_Recipe.stCurrentRecipe.stVolumes.aS3_Volume[2] := STRING_TO_REAL(GVL_DB.astVolData[5].rinse2);
GVL_Recipe.stCurrentRecipe.stVolumes.aS3_Volume[3] := STRING_TO_REAL(GVL_DB.astVolData[5].wash1);
GVL_Recipe.stCurrentRecipe.stVolumes.aS3_Volume[4] := STRING_TO_REAL(GVL_DB.astVolData[5].wash2);
GVL_Recipe.stCurrentRecipe.stVolumes.aS4_Volume[1] := STRING_TO_REAL(GVL_DB.astVolData[6].rinse1);
GVL_Recipe.stCurrentRecipe.stVolumes.aS4_Volume[2] := STRING_TO_REAL(GVL_DB.astVolData[6].rinse2);
GVL_Recipe.stCurrentRecipe.stVolumes.aS4_Volume[3] := STRING_TO_REAL(GVL_DB.astVolData[6].wash1);
GVL_Recipe.stCurrentRecipe.stVolumes.aS4_Volume[4] := STRING_TO_REAL(GVL_DB.astVolData[6].wash2);
GVL_Recipe.stCurrentRecipe.stVolumes.aS5_Volume[1] := STRING_TO_REAL(GVL_DB.astVolData[7].rinse1);
GVL_Recipe.stCurrentRecipe.stVolumes.aS5_Volume[2] := STRING_TO_REAL(GVL_DB.astVolData[7].rinse2);
GVL_Recipe.stCurrentRecipe.stVolumes.aS5_Volume[3] := STRING_TO_REAL(GVL_DB.astVolData[7].wash1);
GVL_Recipe.stCurrentRecipe.stVolumes.aS5_Volume[4] := STRING_TO_REAL(GVL_DB.astVolData[7].wash2);
GVL_Recipe.stCurrentRecipe.stVolumes.aS6_Volume[1] := STRING_TO_REAL(GVL_DB.astVolData[8].rinse1);
GVL_Recipe.stCurrentRecipe.stVolumes.aS6_Volume[2] := STRING_TO_REAL(GVL_DB.astVolData[8].rinse2);
GVL_Recipe.stCurrentRecipe.stVolumes.aS6_Volume[3] := STRING_TO_REAL(GVL_DB.astVolData[8].wash1);
GVL_Recipe.stCurrentRecipe.stVolumes.aS6_Volume[4] := STRING_TO_REAL(GVL_DB.astVolData[8].wash2);
GVL_Recipe.stCurrentRecipe.stVolumes.aS7_Volume[1] := STRING_TO_REAL(GVL_DB.astVolData[9].rinse1);
GVL_Recipe.stCurrentRecipe.stVolumes.aS7_Volume[2] := STRING_TO_REAL(GVL_DB.astVolData[9].rinse2);
GVL_Recipe.stCurrentRecipe.stVolumes.aS7_Volume[3] := STRING_TO_REAL(GVL_DB.astVolData[9].wash1);
GVL_Recipe.stCurrentRecipe.stVolumes.aS7_Volume[4] := STRING_TO_REAL(GVL_DB.astVolData[9].wash2);
GVL_Recipe.stCurrentRecipe.stVolumes.aF_Volume[1] := STRING_TO_REAL(GVL_DB.astVolData[10].rinse1);
GVL_Recipe.stCurrentRecipe.stVolumes.aF_Volume[2] := STRING_TO_REAL(GVL_DB.astVolData[10].rinse2);
GVL_Recipe.stCurrentRecipe.stVolumes.aF_Volume[3] := STRING_TO_REAL(GVL_DB.astVolData[10].wash1);
GVL_Recipe.stCurrentRecipe.stVolumes.aF_Volume[4] := STRING_TO_REAL(GVL_DB.astVolData[10].wash2);
END_METHOD

METHOD insertCalib : BOOL
VAR_INPUT
	start: BOOL;
END_VAR


VAR
	sysRevisionNo: STRING;
END_VAR
sysRevisionNo:= INT_TO_STRING(GVL_DB.stParameter_PCR.sysRevisionNo);

IF start THEN
FindAndReplace(pSrcString:= ADR(cmdIn), pDeleteString:= ADR('#1#'), pInsertString:= ADR(GVL_DB.stParameter_PCR.userID), pDstString:= ADR(cmdIn), nDstSize:= SIZEOF(cmdIn));
FindAndReplace(pSrcString:= ADR(cmdIn), pDeleteString:= ADR('#2#'), pInsertString:= ADR(GVL_DB.stParameter_PCR.density), pDstString:= ADR(cmdIn), nDstSize:= SIZEOF(cmdIn));
FindAndReplace(pSrcString:= ADR(cmdIn), pDeleteString:= ADR('#3#'), pInsertString:= ADR(GVL_DB.stParameter_PCR.solventNo), pDstString:= ADR(cmdIn), nDstSize:= SIZEOF(cmdIn));
FindAndReplace(pSrcString:= ADR(cmdIn), pDeleteString:= ADR('#4#'), pInsertString:= ADR(GVL_DB.stParameter_PCR.solventRevision), pDstString:= ADR(cmdIn), nDstSize:= SIZEOF(cmdIn));
FindAndReplace(pSrcString:= ADR(cmdIn), pDeleteString:= ADR('#5#'), pInsertString:= ADR(GVL_DB.stParameter_PCR.allowableFail), pDstString:= ADR(cmdIn), nDstSize:= SIZEOF(cmdIn));
FindAndReplace(pSrcString:= ADR(cmdIn), pDeleteString:= ADR('#6#'), pInsertString:= ADR(GVL_DB.stParameter_PCR.replicates), pDstString:= ADR(cmdIn), nDstSize:= SIZEOF(cmdIn));
FindAndReplace(pSrcString:= ADR(cmdIn), pDeleteString:= ADR('#7#'), pInsertString:= ADR(GVL_DB.stParameter_PCR.callInterval), pDstString:= ADR(cmdIn), nDstSize:= SIZEOF(cmdIn));
FindAndReplace(pSrcString:= ADR(cmdIn), pDeleteString:= ADR('#8#'), pInsertString:= ADR(sysRevisionNo), pDstString:= ADR(cmdIn), nDstSize:= SIZEOF(cmdIn));
END_IF
END_METHOD

METHOD insertCalibValues : BOOL
VAR_INPUT
	start: BOOL;
	line: INT;
END_VAR

VAR
	CalibrationNo: STRING;
END_VAR
CalibrationNo:= INT_TO_STRING(GVL_DB.astData_PCR[line-1].CalibrationNo);

IF start THEN
FindAndReplace(pSrcString:= ADR(cmdIn), pDeleteString:= ADR('#1#'), pInsertString:= ADR(GVL_DB.astData_PCR[line-1].dateTime), pDstString:= ADR(cmdIn), nDstSize:= SIZEOF(cmdIn));
FindAndReplace(pSrcString:= ADR(cmdIn), pDeleteString:= ADR('#2#'), pInsertString:= ADR(GVL_DB.astData_PCR[line-1].pumpNo), pDstString:= ADR(cmdIn), nDstSize:= SIZEOF(cmdIn));
FindAndReplace(pSrcString:= ADR(cmdIn), pDeleteString:= ADR('#3#'), pInsertString:= ADR(GVL_DB.astData_PCR[line-1].step), pDstString:= ADR(cmdIn), nDstSize:= SIZEOF(cmdIn));
FindAndReplace(pSrcString:= ADR(cmdIn), pDeleteString:= ADR('#4#'), pInsertString:= ADR(GVL_DB.astData_PCR[line-1].tareWt), pDstString:= ADR(cmdIn), nDstSize:= SIZEOF(cmdIn));
FindAndReplace(pSrcString:= ADR(cmdIn), pDeleteString:= ADR('#5#'), pInsertString:= ADR(GVL_DB.astData_PCR[line-1].grossWt), pDstString:= ADR(cmdIn), nDstSize:= SIZEOF(cmdIn));
FindAndReplace(pSrcString:= ADR(cmdIn), pDeleteString:= ADR('#6#'), pInsertString:= ADR(GVL_DB.astData_PCR[line-1].netVolume), pDstString:= ADR(cmdIn), nDstSize:= SIZEOF(cmdIn));
FindAndReplace(pSrcString:= ADR(cmdIn), pDeleteString:= ADR('#7#'), pInsertString:= ADR(GVL_DB.astData_PCR[line-1].netWt), pDstString:= ADR(cmdIn), nDstSize:= SIZEOF(cmdIn));
FindAndReplace(pSrcString:= ADR(cmdIn), pDeleteString:= ADR('#8#'), pInsertString:= ADR(GVL_DB.astData_PCR[line-1].targetVolume), pDstString:= ADR(cmdIn), nDstSize:= SIZEOF(cmdIn));
FindAndReplace(pSrcString:= ADR(cmdIn), pDeleteString:= ADR('#9#'), pInsertString:= ADR(GVL_DB.astData_PCR[line-1].differencePercent), pDstString:= ADR(cmdIn), nDstSize:= SIZEOF(cmdIn));
FindAndReplace(pSrcString:= ADR(cmdIn), pDeleteString:= ADR('#10#'), pInsertString:= ADR(GVL_DB.astData_PCR[line-1].criteria), pDstString:= ADR(cmdIn), nDstSize:= SIZEOF(cmdIn));
FindAndReplace(pSrcString:= ADR(cmdIn), pDeleteString:= ADR('#11#'), pInsertString:= ADR(GVL_DB.astData_PCR[line-1].pumpRevs), pDstString:= ADR(cmdIn), nDstSize:= SIZEOF(cmdIn));
FindAndReplace(pSrcString:= ADR(cmdIn), pDeleteString:= ADR('#12#'), pInsertString:= ADR(CalibrationNo), pDstString:= ADR(cmdIn), nDstSize:= SIZEOF(cmdIn));

END_IF
END_METHOD

METHOD insertLinearMotors : BOOL
VAR_INPUT
	start: BOOL;
END_VAR


VAR

	stIOTerm23: STRING;
	stIOTerm24: STRING;
	stIOTerm25: STRING;
	stIOTerm26: STRING;
	stIOTerm27: STRING;
	stIOTerm28: STRING;
	stIOTerm29: STRING;
	stIOTerm30: STRING;
	stIOTerm31: STRING;
	stIOTerm32: STRING;
	sChangedBy : STRING(100);
    sChangedOn : STRING(100);
END_VAR

stIOTerm23:= LREAL_TO_STRING(GVL_HMI.aCalibLinearPumps[1].rNewPosition);
stIOTerm24:= LREAL_TO_STRING(GVL_HMI.aCalibLinearPumps[2].rNewPosition);
stIOTerm25:= LREAL_TO_STRING(GVL_HMI.aCalibLinearPumps[3].rNewPosition);
stIOTerm26:= LREAL_TO_STRING(GVL_HMI.aCalibLinearPumps[4].rNewPosition);
stIOTerm27:= LREAL_TO_STRING(GVL_HMI.aCalibLinearPumps[5].rNewPosition);
stIOTerm28:= LREAL_TO_STRING(GVL_HMI.aCalibLinearPumps[6].rNewPosition);
stIOTerm29:= LREAL_TO_STRING(GVL_HMI.aCalibLinearPumps[7].rNewPosition);
stIOTerm30:= LREAL_TO_STRING(GVL_HMI.aCalibLinearPumps[8].rNewPosition);
stIOTerm31:= LREAL_TO_STRING(GVL_HMI.aCalibLinearPumps[9].rNewPosition);
stIOTerm32:= LREAL_TO_STRING(GVL_HMI.aCalibLinearPumps[10].rNewPosition);

IF start THEN
	FindAndReplace(pSrcString:= ADR(cmdIn), pDeleteString:= ADR('#1#'),  pInsertString:= ADR(stIOTerm23), pDstString:= ADR(cmdIn), nDstSize:= SIZEOF(cmdIn));
	FindAndReplace(pSrcString:= ADR(cmdIn), pDeleteString:= ADR('#2#'),  pInsertString:= ADR(stIOTerm24), pDstString:= ADR(cmdIn), nDstSize:= SIZEOF(cmdIn));
	FindAndReplace(pSrcString:= ADR(cmdIn), pDeleteString:= ADR('#3#'),  pInsertString:= ADR(stIOTerm25), pDstString:= ADR(cmdIn), nDstSize:= SIZEOF(cmdIn));
	FindAndReplace(pSrcString:= ADR(cmdIn), pDeleteString:= ADR('#4#'),  pInsertString:= ADR(stIOTerm26), pDstString:= ADR(cmdIn), nDstSize:= SIZEOF(cmdIn));
	FindAndReplace(pSrcString:= ADR(cmdIn), pDeleteString:= ADR('#5#'),  pInsertString:= ADR(stIOTerm27), pDstString:= ADR(cmdIn), nDstSize:= SIZEOF(cmdIn));
	FindAndReplace(pSrcString:= ADR(cmdIn), pDeleteString:= ADR('#6#'),  pInsertString:= ADR(stIOTerm28), pDstString:= ADR(cmdIn), nDstSize:= SIZEOF(cmdIn));
	FindAndReplace(pSrcString:= ADR(cmdIn), pDeleteString:= ADR('#7#'),  pInsertString:= ADR(stIOTerm29), pDstString:= ADR(cmdIn), nDstSize:= SIZEOF(cmdIn));
	FindAndReplace(pSrcString:= ADR(cmdIn), pDeleteString:= ADR('#8#'),  pInsertString:= ADR(stIOTerm30), pDstString:= ADR(cmdIn), nDstSize:= SIZEOF(cmdIn));
	FindAndReplace(pSrcString:= ADR(cmdIn), pDeleteString:= ADR('#9#'),  pInsertString:= ADR(stIOTerm31), pDstString:= ADR(cmdIn), nDstSize:= SIZEOF(cmdIn));
	FindAndReplace(pSrcString:= ADR(cmdIn), pDeleteString:= ADR('#10#'), pInsertString:= ADR(stIOTerm32), pDstString:= ADR(cmdIn), nDstSize:= SIZEOF(cmdIn));
	FindAndReplace(pSrcString:= ADR(cmdIn), pDeleteString:= ADR('#11#'), pInsertString:= ADR(sChangedBy),  pDstString:= ADR(cmdIn), nDstSize:= SIZEOF(cmdIn));
	FindAndReplace(pSrcString:= ADR(cmdIn), pDeleteString:= ADR('#12#'), pInsertString:= ADR(sChangedOn),  pDstString:= ADR(cmdIn), nDstSize:= SIZEOF(cmdIn));
END_IF
END_METHOD

METHOD insertMethod : BOOL
VAR_INPUT
	start: BOOL;
END_VAR

VAR
	iRevision: STRING;
	dCreationDate: STRING;
	Rinse1: STRING;
	Rinse2: STRING;
	Wash1: STRING;
	Wash2: STRING;
	Rinse12: STRING;
	Rinse22: STRING;
	Wash12: STRING;
	Wash22: STRING;
	Rinse13: STRING;
	Wash13: STRING;
	Wash23: STRING;
	Rinse23: STRING;
	soakTime: STRING;
	agitate_1_Time: STRING;
	vialPrimeVol: STRING;
	vial_2_4_FillVol: STRING;
	vial_1_FillVol: STRING;
	airDryTime: STRING;
	agitate_2_Time: STRING;
	vialsToFill: STRING;
END_VAR
IF GVL_HMI.bNewRecipeButton THEN
	iRevision := '1';
ELSE
	iRevision := INT_TO_STRING(GVL_HMI.stRecipeInfo.iRevision+1);	
END_IF
dCreationDate := DATE_TO_STRING(GVL_HMI.stRecipeInfo.dCreationDate);
Rinse1 := INT_TO_STRING(GVL_HMI.aSolventAndTimesRows[1].Rinse1);
Rinse2 := INT_TO_STRING(GVL_HMI.aSolventAndTimesRows[1].Rinse2);
Wash1 := INT_TO_STRING(GVL_HMI.aSolventAndTimesRows[1].Wash1);
Wash2 := INT_TO_STRING(GVL_HMI.aSolventAndTimesRows[1].Wash2);
Rinse12 := INT_TO_STRING(GVL_HMI.aSolventAndTimesRows[2].Rinse1);
Rinse22 := INT_TO_STRING(GVL_HMI.aSolventAndTimesRows[2].Rinse2);
Wash12 := INT_TO_STRING(GVL_HMI.aSolventAndTimesRows[2].Wash1);
Wash22 := INT_TO_STRING(GVL_HMI.aSolventAndTimesRows[2].Wash2);
Rinse13 := INT_TO_STRING(GVL_HMI.aSolventAndTimesRows[3].Rinse1);
Rinse23 := INT_TO_STRING(GVL_HMI.aSolventAndTimesRows[3].Rinse2);
Wash13 := INT_TO_STRING(GVL_HMI.aSolventAndTimesRows[3].Wash1);
Wash23 := INT_TO_STRING(GVL_HMI.aSolventAndTimesRows[3].Wash2);
soakTime := REAL_TO_STRING(GVL_HMI.aOtherParamsRows[1].Value) ;
agitate_1_Time := REAL_TO_STRING(GVL_HMI.aOtherParamsRows[2].Value);
agitate_2_Time := REAL_TO_STRING(GVL_HMI.aOtherParamsRows[3].Value);
vialsToFill := REAL_TO_STRING(GVL_HMI.aOtherParamsRows[4].Value);
vialPrimeVol := REAL_TO_STRING(GVL_HMI.aOtherParamsRows[5].Value);
vial_1_FillVol := REAL_TO_STRING(GVL_HMI.aOtherParamsRows[6].Value);
vial_2_4_FillVol := REAL_TO_STRING(GVL_HMI.aOtherParamsRows[7].Value);
airDryTime := REAL_TO_STRING(GVL_HMI.aOtherParamsRows[8].Value);


